(* CoDeSys 2.3 project: cy-wg-021-003.pro *)
(* Title: cy-wg-06 - ClevergyAS *)
(* Author: Andrea Ravasio *)
(* Libraries: Standard.lib 8.11.10 12:37:48, Util.lib 26.9.14 11:12:46, Visual.lib 8.11.10 12:37:48, WagoLibIdent.lib 25.2.13 13:49:34, WagoLibStatus.lib 8.11.10 12:37:48, SysLibFile.lib 8.11.10 12:37:48, SysLibRtc.lib 8.11.10 12:37:48, SysLibSockets.lib 5.5.11 09:22:24, SysLibEvent.lib 8.11.10 12:37:48, SysLibPlcCtrl.lib 8.11.10 12:37:48, SysLibCallback.lib 8.11.10 12:37:48, mod_com.lib 8.11.10 12:37:48, SerComm.lib 31.5.11 09:06:48, Serial_Interface_01.lib 22.4.13 12:50:14, Modb_l05.lib 13.5.15 10:30:08, Ethernet.lib 8.11.10 12:37:48, MBus_03.lib 9.2.13 17:51:58, WagoLibModbus_IP_01.lib 26.5.15 11:20:08, WagoLibMBX_01.lib 20.3.12 16:32:38, LON_01.lib 28.9.12 14:05:10 *)

(* PLC configuration (modules and I/O channels)
0750-9999/0545-0008 8 DO/DI Generic [Type_34_8_Channels] node 0, in %IB56 out %QB32 {INTTypePAAssignment = PLC; INTTypeModule = plugged}
  VPN_ST2 AT %IX28.0 [BOOLOnX_I] I 1: Digital Input
  LAMP_AL AT %QX16.0 [BOOLOnX_Q] I 2: Digital Input
  KEY_QE_ST AT %IX28.1 [BOOLOnX_I] I 3: Digital Input
  CIR03_EN AT %QX16.1 [BOOLOnX_Q] I 4: Digital Input
  CIR03_AL AT %IX28.2 [BOOLOnX_I] I 5: Digital Input
  CIRD06_B_EN AT %QX16.2 [BOOLOnX_Q] I 6: Digital Input
  CIR03_ST AT %IX28.3 [BOOLOnX_I] I 7: Digital Input
  CIRD06_A_EN AT %QX16.3 [BOOLOnX_Q] I 8: Digital Input
  CIR03_AUTO AT %IX28.4 [BOOLOnX_I] O 0: Digital Output
  AT %QX16.4 [BOOLOnX_Q] O 1: Digital Output
  CIRD06_B_AL AT %IX28.5 [BOOLOnX_I] O 2: Digital Output
  AT %QX16.5 [BOOLOnX_Q] O 3: Digital Output
  CIRD06_B_ST AT %IX28.6 [BOOLOnX_I] O 4: Digital Output
  AT %QX16.6 [BOOLOnX_Q] O 5: Digital Output
  CIRD06_B_AUTO AT %IX28.7 [BOOLOnX_I] O 6: Digital Output
  AT %QX16.7 [BOOLOnX_Q] O 7: Digital Output
0750-9999/0400-0008 8 DI Generic [Type_1_8_Channels] node 1, in %IB56 out %QB32 {INTTypePAAssignment = PLC; INTTypeModule = plugged}
  CIRD06_A_AL AT %IX28.8 [BOOLOnX_I] I 1: Digital Input
  CTL02_ST AT %IX28.9 [BOOLOnX_I] I 2: Digital Input
  CIRD06_A_ST AT %IX28.10 [BOOLOnX_I] I 3: Digital Input
  ALARM_PB02 AT %IX28.11 [BOOLOnX_I] I 4: Digital Input
  CIRD06_A_AUTO AT %IX28.12 [BOOLOnX_I] I 5: Digital Input
  CIR01_AL AT %IX28.13 [BOOLOnX_I] I 6: Digital Input
  CTL01_ST AT %IX28.14 [BOOLOnX_I] I 7: Digital Input
  CIR01_AUTO AT %IX28.15 [BOOLOnX_I] I 8: Digital Input
0750-9999/0400-0008 8 DI Generic [Type_1_8_Channels] node 2, in %IB57 out %QB33 {INTTypePAAssignment = PLC; INTTypeModule = plugged}
  CIR02_AL AT %IX29.0 [BOOLOnX_I] I 1: Digital Input
  CIRD01_B_AL AT %IX29.1 [BOOLOnX_I] I 2: Digital Input
  CIR02_AUTO AT %IX29.2 [BOOLOnX_I] I 3: Digital Input
  CIRD01_B_AUTO AT %IX29.3 [BOOLOnX_I] I 4: Digital Input
  CIRD01_A_AL AT %IX29.4 [BOOLOnX_I] I 5: Digital Input
  CIRD02_A_AL AT %IX29.5 [BOOLOnX_I] I 6: Digital Input
  CIRD01_A_AUTO AT %IX29.6 [BOOLOnX_I] I 7: Digital Input
  CIRD02_A_AUTO AT %IX29.7 [BOOLOnX_I] I 8: Digital Input
0750-9999/0400-0008 8 DI Generic [Type_1_8_Channels] node 3, in %IB58 out %QB33 {INTTypePAAssignment = PLC; INTTypeModule = plugged}
  CIRD02_B_AL AT %IX29.8 [BOOLOnX_I] Ch_1 Digital input
  CIRD03_B_AL AT %IX29.9 [BOOLOnX_I] Ch_2 Digital input
  CIRD02_B_AUTO AT %IX29.10 [BOOLOnX_I] Ch_3 Digital input
  CIRD03_B_AUTO AT %IX29.11 [BOOLOnX_I] Ch_4 Digital input
  CIRD03_A_AL AT %IX29.12 [BOOLOnX_I] Ch_5 Digital input
  CIRD04_A_AL AT %IX29.13 [BOOLOnX_I] Ch_6 Digital input
  CIRD03_A_AUTO AT %IX29.14 [BOOLOnX_I] Ch_7 Digital input
  CIRD04_A_AUTO AT %IX29.15 [BOOLOnX_I] Ch_8 Digital input
0750-9999/0400-0008 8 DI Generic [Type_1_8_Channels] node 4, in %IB59 out %QB33 {INTTypePAAssignment = PLC; INTTypeModule = plugged}
  CIRD04_B_AL AT %IX30.0 [BOOLOnX_I] I 1: Digital Input
  CIRD05_B_AL AT %IX30.1 [BOOLOnX_I] I 2: Digital Input
  CIRD04_B_AUTO AT %IX30.2 [BOOLOnX_I] I 3: Digital Input
  CIRD05_B_AUTO AT %IX30.3 [BOOLOnX_I] I 4: Digital Input
  CIRD05_A_AL AT %IX30.4 [BOOLOnX_I] I 5: Digital Input
  ALARM_PB01 AT %IX30.5 [BOOLOnX_I] I 6: Digital Input
  CIRD05_A_AUTO AT %IX30.6 [BOOLOnX_I] I 7: Digital Input
  AT %IX30.7 [BOOLOnX_I] I 8: Digital Input
0753-0648 LON-FTT [Type_55_1_Channels] node 5, in %IB52 out %QB32 {INTTypePAAssignment = PLC; INTTypeModule = plugged; DataStream = 1F8B0800000000000400ED5D7B6FDACAB6FFFF4AF73BCC41BA47AD141A0C84909C245B144C83368F1C1EE9AEDA0A393080778DCDF12369CEA7BF6B666C63E3F18B47D2504B5BDDC41EAF596B66CD6F3D66797CF5C7CFA5821EB16EC89A7A9D133E147208AB136D2AABF3EB9C65CEF24225F7C7CDFFFECF555B535BAA89F599; DataStream = 34C1081E528DCB9F867C9D5B98E6EAF2F4F4E9E9E9C353E983A6CF4F8B858270FA57A73D982CF052CACBAA614AEA04E7DCA7A6F14FE5D09DAECD7569D982C61785CB42E1F21CFE3DBB2C089785CA65A10C3F72E82F79D69596F83A272A78895553D2F1B82DC9AA3C160B173934C0CAACA14D2C7ACB0401EBDA92FCBECED5A6; DataStream = 53F4AC593A9AB02B68817560B08B2D5D539BB2BE7C0252F7EEA85CD0AE06D223BE93CCC575AE7EF9ED936C7E9B3CE70B4235FF3447EF1AD8C0EA7F2555437792820D5397D0BDAC2812EA482AD09751AD20D4DF7F6BF7BA39D4D1A69682BBD6F201EB403C07A38B1019DF8EA4FFE83DFC8D27A641AF6D5EB52FC2E5215EAE14; DataStream = C9C4AD29213E93B1EEDE83BB64E85AD39B4201F1FEBB3AB5EF7B9E184CB415BE815BEC87E7CE9FF8995C27FFF35C6DA953FCF346B83A653F5CBE4E231873992653763368DE0D556D8A9964EB07E94DF7116E537F939E2ECF655552B84D7D37DD475A465B9BFCC0D31B53B730C8E0FCE96900D336954C4D7F76DBACAF789AF5; DataStream = 5644AD24E5662629066DE65E715B7530996836DD64287D7FBBAD6C0DAE6B1668232CAC4B5556AE73A4F31C3AF50C08369F34FDC7BDA4CBD203289A775236EE796EC569CC765A13AD39AEF65C1437D5C7A342E4A65F8762F588A34BDDFBE1587BF87BACE3FF58B0F842B469AD51EAA3DC779A069BF894C6DB94AB4D89342A85; DataStream = 5625D7ACA0760921DA455B26D33046545607589D0EE5259D5AEF9FFE76D24F5F3BCF9F9BEDFA7882E547EC69EABDB221FC9D2E6BBA6C3EAF8577AFF85A0EB0FE284FF0F01934AF36F9A16A4F0A9ECEF114B4D173C7F74843D6011960206F5AEACA82495D5FF0B30C2670264FC8DCDC74351598F05EF135AD6BEA4C9E5B3A35; DataStream = 31B04A565837656C6C0E6ACB70BBDA5096CDEBBEC73E3E9B7820FF17DF94AE4EDDDF9E557F1ABEEC7F594428452142699F8800AE8769190900411BD82D63F1C06DF9CBC341318383E470D0B3CCB7850795A3C183F3283C38DF1B1ECC6405131721897BD084B67DD234DE3D709BEE110F5C458F07048764023C38CBF0E078DD; DataStream = 03A1783C78508EC283F25EF120B98340D63931FD495C8475DB5F1E142A19281CB193503C3F1A54B808A4A1D808B1A8A1B0575458694920819AFE3B2D49D0B06EFACB03C2790608C7EB25A40D1A0277D619C75896AF4E79D9EBED52DAD109EABC1092A1CEA74C51D345792FEBA625296866A913B65AD0830283BA99794E9546; DataStream = 8E58AB591E3919FEFF7A7964686E278785581B10249EC012B8EAB0475390268314A666B465660BD0AFE61CBAE26529653642AF975286D62C519C021A8CE499E50C19DE1032BCBE979812188E27B75C8DCA2555F7964B3241B5C8F25DAE92000351C4014EEA34786967C8705CC8F0F67C86E3492855AB51D050DD1734488AA4; DataStream = 2F93A0428D344C880936D10C0E8E0B0EDE9CA350BCC8E0E0907090DC4BC810E12811E1ED3908C70409515985EADEB20A24ECC789928DCA33C929E0849060D3CD20E1B820E1ED39094703084221CA49A077F703098B4769325E6AD344B0D0B8FD3C86494E9152F090CFD0E1B8D0E1ED390CC211C1C359243C9CED2DDD0857C6; DataStream = 89528D041B6A1393344C9A6EB46967C0705CC090B90D192EF87101FC853B4D5613EF4364C07094C0F0F63C860C190E8F0C99C7F0DB0343E631BC5E3D53142C5CEC0D158C27D99C2C92A042BDD920A820AA49738F36E50C138E0B1332672103051F287CCA40E1B70785CC51C87624D820F9BD05B22991ED48FCEEE8F0F65C86; DataStream = 6C47E280F905820D5972E1B74785CC67C84021E03064DB111930BC3D77214386C32343E631FCF6C090790CD9D90B6C90FC672F14B3B3177E7B6C787B4E4376F6C20B9CBD90021AB2B3178E1319DE9CD7909DBDF012672F244486ECEC85E34586B7E73364672F1CF465EB849890BD697D9470F0E61C85637AD1FA578483E45E; DataStream = 4286084789086FCF41382648F845CF5E480809D9D90B4709096FCF49381A40F8352B1D3D672F244486ACD2F168D1E1ED390C59A5E3CB9CBD9034DD98952E1C2530646E43860BFCB3173260F8AD81E1ED790C1932BCCCD90B1930FCD6C090790CD96BD681B31792E61EB3D7AC8F12133267210385E0D90B1928FCD6A090390A; DataStream = D98E041BA4E0D90BD98EC4EF8E0E6FCF65C876245EE0EC852CB9F05BA342E63364A0C03F7B210386DF1A18DE9EBB9021C3CB9CBD9001C36F0D0C47EF3104EE18EB5B713C5F9DB635B523E93F7A0F7F036BF4EAC635E3E6EA1F5FEB8DDAB0F6F5EA8F9F4B053D62DD006AD739E1432187B03A810153E7D739CB9CE5854AEE8F; DataStream = 9BABBA644A8A36BFB96ACA0A462D03FE67621D4FE1911C6AC0CD7B974499D020CDC8145EE7C8BFF0B7A62F25D36D54216D3AD2DF9AEE792E87EE2473719DAB5F7E23B0A54B4B4AC640EF7E562BEFBF81089F61488C6F84A2F16D30AC751BB57EE3C3F0CB1D3C4971EE3A17028439D4C733E0579DE0C856F47D4CF28225F053; DataStream = 3C154AA7C582504442F5B258B8148AB99B4DB8A6AC70AFA28F92618FC00056EAC4FC5AF99E43740983F83944D1F33A775ECA21024BD7393AB0F6911070EDD1640F131C0309C5F160D81FD5874C52181A184D79C29EA4583783C7C989123944B48CB09F43235586CEFEA998FF6AA98F92224F9161EA30B1D08DA159FA04FF73; DataStream = 6EFE8B2F94877D51B596C8214FB81B9B64EE7ECA4B6B4945019061BFF382234C3F5C0EB13BEAF0A470451FC873D5562C5B144792996788900A4F193944B8C36C31D8437A46403146A6916AD05E40A7E63017464B35F11CEBB4AF963198907768E81F6B39CFCE4A678E78B4279E70A3EEA0F5A92B36C6ED5EF7530EF5663303; DataStream = 9B945050609911219DE19A47DCA24F5CBBD5A125B2211D91578C358B3B7121B295F89349C98D5D72E1522E6545910D3CD1D4A991484E98E9AFA5F55A72175003B402AC3CD104244DA7A0E3065F8C56AFBB66FF8CC7FE9468B94B83317CE630ECE090DB49C2F55F5CF35C7478AE3112C8248F01F09AFA73D4DA8F649AB0633A; DataStream = DC961C6E793D24D5A5C1422314932853A9E4C1815229201F3502113A35B8EDF5E3046444029AE4C24335FF209BC8B299478078CC413AECCAF10FB09C12192A5B218350091375D371A06ED436F6C9362DD6838ACDBCAA4D71D49A4AA49F861ABE940C4E3F07D052C1A3A4C25BD2D18FB2E94ECE864036F8694B495679EC7F6C; DataStream = 0D9B31FA36B51F0E67DB9D28D634B55542E7888A00FF786CA22DD0B957A0E2B923521794614B8154FA68B83854CF541A69A511A21C10A2EC0A51F60AE131AB80B768429AC48B72CEB7A4D42644C842C540DA0C91A6324E6644B79668A84BAA21D190873A0B7ABC5C55EE42F939B61F0F178D3680D183C94A0BE62940A17876; DataStream = E687BB342070C1453A9B4CB864AC8557057700EEF3EFDEA5C458F8A46BD66A67C89EAFC2217BEEEB6167008B4361BF4A6D85BD0F9AA660493D046C55D62A047D6EC9BF411F4D00C26CE859F3DFDE74303E46AA6540DB998C95E996A25894449428719174664A3253E203E09D2DC99C51D94D25F9A6651B83B39DCB6D03BC65; DataStream = 2EC8A6C08445E81A1771C206472870235E2039D622D1273DE66F239B93E34E2B15372FB4026229A4DAC171287FF7AE50272359F66524D94994DB26249DA7EDF8F57CFF3949D6832F252908DC9CE4205492B094E49AFBC88C246B169E90AC1C3E09D175919B701492F74A9E9A648660ACCDC636B9F054846D900E2DE0002B78; DataStream = 62520BAF4447E909B293864D6CCC88ED2D034B32931159BE6DB391D2547739DB5B56DF86809044EA449757A6C635C8890287A987C4BE39AFE9BAF4FC55A87C27EADE643334D390442E23CCB64AD71E2FD96A31E8231EBC769FE20958EBF76B5F62E4A3D0C308D8885071C4637C006B42054D16920E0E0ED6132489E9EAA8C3; DataStream = 03096D0F01530FCA15AB01E136878433976CC9D46F6BFDB5C045AEAD7525FE2A9C7DDF583361E8C8925DB541BDD55A0FC5F6468BF6F36F4B9A2674C684F279B95AAA94CFE362337B18FE3DAA353CC3C045464E8CB6217DD935D2CF662A0F7A4B641CC6A52DFD80584C133A275EB37B7544624133F1768867FBE662BFF0C3D0; DataStream = 8785CEA8D508411F2EF8B80F6D0B3E2C901ECB5347B620F65410D3BEC3C638A1E2EFEAD8BB127E0D604DB26CFA0B0537958D9150B03A3717BB8700B6FC0EB9F00110BB48285F14AA79C149AF38CFFC7299525290B09F54E9FEE3B8F84D8750A9B80E66DAFD873411FA0E302B78B6F884750D4AB5E40D91307A04E738DAF70B; DataStream = 09F9E831839CCD4AE242CB8FF2D4921444162C5DA77BC819337609C54278EA28C82B3C50D84FCE203C3119C3AF90925FE130FC1693F25B4CC96FF130FC9692F25B4AC96FE930FC9693F25B4EC96FF930FC9E25E5F72C25BF6787E1B79294DF4A4A7E2B87E1F73C29BFE729F93DDF23BFC938ACC627EBB9AE0D3C5B7D65F0BD; DataStream = D89EF58B57C66121C2D0C5F12E1CC8E825066521C2EAC5327F200B9818A185081318CBFC81CC6162B81622EC612CF307B28D89B15B88308EB1CC1FC85026067221C252C6329FD86AEEADEACF8908DC2C0C298847F493435BC403EBEF1539DCBB1B40CF58D24FD05253CDC5099A4ACF2768A159E48AAC5A263E41AC203861D6; DataStream = 3479E6AC542055FE9CCDA12F58E2473CDE1C5A50CC67FA58543AB0E895384D3A3055FCEA88D121039A267EE506E54B46255CF768830309535A27CA246E31749828DC487C2A45563CC0ED0389517483EA5B50EC34729479722C28917041C8FD03497276E16A175D9C3BD7C82E6D3211FA455B1C5C9E01039914F2700B876CAC; DataStream = 8ACA61795E6FD8257FE3C9930BEB1DFBAABBF543BF14B3FD963DFD728C0B5C07C998B735BBFE2345C2DC7926225F1E1448711F7ADD1C7998C03BAE2147BC74097222F0CEF9F12DF7A9D8AB8721DB1E69DE8ED02821B6FD11BA61C51A25DEBBA7F52454FDC7642BCC574E522AFA3C86927FB19921DB6FACA624B26E6DDD5FD4; DataStream = 26AAE476135E61729E54C4955DA83456F023569254CDB8A54DF4897849B9656CFE6EA3A45DF9BA0B97B8FA422FF911A0E8DEA7A9A7E16E68513D1C9BDA98E06C94DECAEB4ED144B20C02B6362CC7CACB70B64C71F69EA4D84340B6CC03D97BB67716BB23C9DFC6B177DE3676C05DA82DBF08D472654EB195C3055A2A192D93; DataStream = 8908C55E16565910131DB784692717513951CC1B085D042EA8BECDD845E0C2E61B0C5EF8C5436F347AE19700BDE1F0A5C8DF834F15BFEC1BCD2E2E3C33E4BE0A9EA6A2891BF82FBDB4F6F6F6B9D7C432FF4F9197E061A730B49EC712985B7EB916F31C6D1AAF6B74234621855E46F8C794F46E06788790DB5FCE6B3B9F17AE; DataStream = F9A5B5962BCD90C3E2D32445F2F07C204A5D91F3CFB07EE2D4F31CBE38B28FA5E9E967F0BD8940B4F3D85249CE2B464FE395199311753595565793A95BBFA778F8632E5C2113D46AF971869B97038143ABB45C9059BF57B5AE09DDBB4EBA8E941D686F7F940CC4CE63CF692CBEE3245A8D1397F22F943078C12C814D987716; DataStream = 4EB1CC0DA1E327C41F42738DB4BFDBA8105AF375171E429348754745F46C1E15D7BB4717A50DC9B74E48124DF4BF4254F12AA2FDE2CD4C91E6C9CDDCD168636CB1869DB3CDB71A7488E23722B98A27332A7CDEF7B0952A2413C251E73D48B25E432F5FCAD1900D4264BA8B1C539BC6AB9473F42C33AFCDF2D42B33769142B3; DataStream = 4CF2821923F42AC51DBD1556F313599F58F24E7AA5019DB14DE7550A3DEC3931D8C9897B98149BD2AB147E74F06421A932749C9F4996B2D3CC2C5D5A634AEB558A419A184F1FA4C90F1047562C7DA7F999D9B4C636AD172AFBEB3D623DAF4BEA3C29F3DC905C032A634AE5552CC908ECEA1EA4B00899438A11634144F2EEAA; DataStream = 9E7A7D7065C12EAD43AE8F188B3252098DBCA9E5975832922F9090D921C4C84E8B4DEC552C4B5D5B2E2DD53EEAC048B9F0B9724D80E201167D721BD384BEF1146C8C32CB9BC91D31AE30448E31A134360FE687C595173A72E46535BF221C92C3877690C915672CAB6387E0ABD81B7612711E4CF92EF22894CA987F78E7216C; DataStream = 4C47522DC0B489A69ABAA624649D9B9359524A639BD22B452D2BF0C9D8D6FD0E92802A3935392F6F68980CC468EBF23429788589E19079150BD3C72B4D37F34BC9F8B18B183A253326645EC5AA381CC9EA3C4F3E90B58B2CAB352DFAB1AD57B1295E81884DD8974084D6AB5815BA19925735539E3DE7A7E9427DAE546C0B84; DataStream = 111C1F36EE8FB12A7D6CF0DFF74DB470E01EE0F172A5E0E89DD32D8EE8AB22AF69714B21499FFA239E26786D83BBC5E679FE10A76FED90E85FBF834D3FA2B9455AD5B01FDCC83FD252179655C507D9355C97AD84561B6DEE1086971AD993E2BC23F19165DC3726E8FFE8914896A238E56BB17A35D8E54C61FF615351678D6C; DataStream = D67F841D3F1573D8882B286D4BCFB7DBF17C153B3DEE6C119C252C7C299E577CE7D114CF4B82BBB5483ED942F61E68EC92FA1D0BCFA75CFC83E14C7B31EAB58B29064F1C1BA88E1543B6926C31D25D1EFA154AD33310559F2273E7FCF6BE5647CB900304C2CE18F37FF3326A8A5DF2115B3AE5D0D9376EAE3CEDFD7FA1F597; DataStream = 1386D2DC3EEB67BDC17573C52AEB7C0979642FE1A044CDFEB83B6AE7505F7AA26DD8109DFAA90C0875D594250549930989BD744CF6AEB9E47A7762773CEC8D0762B79180D213D9DF8D21D517EB62EB5EF4721964B2AE680646920AE02E3D62FBE8312ED97ABB3710C7CD56DB47B11841718A892D8CA7D910DBE23048BA1420; DataStream = DDA74776029B53FA491A4D7F76BE27C0A5DE68C1100C7BFD2FB0EE7A7F8EEEBCC4CB41E2C0B2B64C3955E37ECD4BF52C866A8A69DBA0CC0ED83BF5683457BD2B5EF576CF0D4CABDD8304DA4DCB424C72BCE90CEBC8B0A88060864208FED51441C43F03641AEE4C2A9AF6831CF91B4789CD25A515A5D8A2AE6B3A22A770AEB0; DataStream = 4ABC9650351CB0A16FD65AED68CD76494E37988EE654ECF7A3D5DA3F94B28AD6B995F0B11C751B62FF33A9A38A526A9765A2CF300AA744036346A3D5DB6439A8D67E96C94B905344F3285C8AC35647EC8D869B642B01B29F65582D4FC8A07837C10813F643887E6E751BBDCF9B34CF0334370E6575138C5CA2B5D1F0769364; DataStream = 354892AD6666A83413747645C266CC470CA05AAF8B83014C59ED7E43C92E6200E3013F6B80A4628F7B2A02901E88E29FE356F7BED626DBF69E055108CE99DDFA73ADC5F53AFDF73DA48464D8736E638FEF1D133F0BA3D594F870EEFC2E402B3177826BEDF1AD580315F7C35070F16C929C699A194AB2D9EB0D374906D77903; DataStream = 3F58737ABC20F9A01791F01D99654965AF29BC0F21DE103F8E3EF9690761A9E5A16A31D613116F759B3D3FEDE0040F9E0DF021D3333EF832188A9D6017C1F5395CD8674B23D94076AD410851D0C891C8D3CC7C104D7C642570F155305DAA7D88523219EABD2EF95A9A4F71F3413C243D4D31DD4286AEB4D94C91552E1600C9; DataStream = 5EB3D96E757D2E493EA87FAC389414D7CA6C5255F2A53F18F9A5F40CCB174DA1A5A951A93C1B260E0C2140E785A44F9F24B277C2AE858938EAFED9ED7DEEFAF8092AAF63DD3DEF54D9C3286D704A916B8527E41B96D3B04EE31D81AE863629AF486641E55A0342B24766ABD11AD263613797B3EAB294926CADDDF1D28DF20D; DataStream = 869A2929A74E2D012D047D24BE35ED4F40EF481A4753A12B5A6106C6DE404E63982F72069D895509D0266CD486BDE178705FA73C09D14E45242FDC0DF20DFAC568E722923E775B64837E29DAC3B08BA3C16ADB05D26CD2142CE9881BF203F936D8ED766708EE7FDF3F3C416888221F363A5EF2C5688783915FC8F3450AF66F; DataStream = 5B9F6EF9FC73BC8FA80EC204F075508CF145B8031437F201C50C3A227CC271631ED0488E9D0A1993D8E10E30CDB1AF21B463473AC87770A9360109364129CCD168F509491F419EE30F0401D5F2C989DEF5C500E1E0A22484F33A261F1B9E829BAE590FE0AEBFA3F50FEF137533EC7FF4E1BEC00B013C7D80074C10C6D0E8F7; DataStream = 3B1CC07E873FCC3F9C8091D165F587028102417023C2C491AE07A3BB7B5FD7C155EB178FEC7053573CF9280EC5C130308CC1C51BD24FBA19A37DF1A62DB8967DFD2D592A0E61F551D63595BC6F02B84D4C13560DE644B0178821B49B2CF8B187CD82D8BDAFF73A77E34EED2F1F07C145EFE3407A508923A980D55859662261; DataStream = 3BBD6E6BD8EB5343ECB37B9C70C42FAC6B53611AB11E66E4691FB55697CC9ED8F7797B454E8E827CD11749AB95E2B85DA10125A15D1BC2BF10FCF5FCF17A90F51E44943AA3153B2A417A413E193DF00169A2228EE2E75ABFDBEAFA228D5231598856B543B4C03BF22933447749F29F6DED8914D1B095B2DA78C79E4BB32DDE; DataStream = 8BED7170BCDD5B5C13E1BD1BE5F5B9EDB8C6C07B37CA5FBB05D3B29558A5683FAD2DCF301A48330CC4A85DA096CC40EF3ED6EAE47060F7908222173CEF363C91A04DB863DFD17E4ED44929AC9362B4BB46890E3CC680D9E300FD7218FD52B4BF46E90F99413B6DD2DAC0770DD95829D2F3FB602F6761BD94A39D36DACB1DC0; DataStream = 13E5FE04D16D893AC99C4D004F44080956048EC384AB84755B8976E568376133520D235A8D76E3C278EF0FBB274C07E057D4200A8550852BC4387AB46F4A5E6158E02C175E37A1A32654383E5F2CD4117628D6055E664A8975FD7F27C03A91D664DA2F4ED1CD0F1D2FB547B8E21605F129F7FA9D5A9B9315373CF4429E6DB4; DataStream = 06B58F6DB1118D7AAC30C8E1CC79D3884B7074D7A80DC9CE7A6D381A44A3E01DD64992C925EB941A86501E88ED267584A231D0CEE549BE239EA258ADB56BFD4E34ECD9F2DBEF5191A382587113976C5FBCEBF587E0610CFE8CC6B99E5332163943BD7BB0FEAD86188D693EDD09A12476C95447A356DFD6383625318AD7EFDC; DataStream = 73D90BA2529D86AA49F4A7DE166B7D8EFA0441C947D32EFF8B201998660ED6D8A3C874875613C9CEE9585CCA9426ACBF61ABF9C51EDE06076778AB72BB3EB8CB95B3C9E4439219CD37915A4FE4D67A72BBEAD4BA2392061DF6FD715B7091053B2050452B2BA23AE88B9D1EACB840079C3D27D681A75A8D54A8D0B41E136326; DataStream = CF2D1BAC57CC29A1DF61E4767BD7EF7DEAD7FC931F5C8E4C9F680D56DEA9C1A23569E89DBF308B6B635C3DEB8B03D1BFF5C159AD3FF1C402EAAC3377DB01248C5CC041D2C105CCA400089490A2CD23396DF77CFE3F27966C6B12C4AC0B771ED6A95EB2C338A8DF0DC90DF6CDB190AEDABD5A833B019C5D2B4BA59D4D2C5D07; DataStream = EF42213BA3D214FAB27BFF805A331F374F92811692C2623FA2DFCAF30934900DF4242B24A635C0A223DD52D9DEADAE2DD9E3E4B57D92BA5F3FFF216CC4475D1EF39C48F416E8C4703F74395BD95573FEB1A5A549C4EC4BE43BEF4C2BC0C7825121697F72C32B96F7512ADA13C47F18816D8A17EBB6D61E72E5E2997EE04B8F; DataStream = 166D3DB40F782ED3D10E1D50B0DFB53EBFF3208E8D54C5D1C0B0BEC36C7B374CF18A1C3463CBD1A01DA9F8A749960E7575B595E311BE239B3C76D11FF17D4F600518B4FC10EE9EB007D003791BE0046173F2E13D59CD71FAB039F94B0BFCDB078CFEF91F4B33FF254F15CC7E911D03F68BCDAB7D956C094D26786532A5B7B5; DataStream = E404692415F0241B4C1B88CE004D79AE6A3AA884AF5B1D9B96AE1A841287BEAD913393242AE818D12F92CE7CDD85796B43F18E3BFCE584AE77D976BDED0A33BEC3FD18E67093A82181CB5D67E68AA41525CBD428010223E4336CEA1C93BD73F30963D597FF21F93BAEA9A19DD646C35E101DB0442B263455E1161AD1276FC5; DataStream = DA30DA0FAFADB9C8DB503C017658CAE789D454F3EB4828F94EBFFB69FCB9DFF1D730716AAF344D89E5B5DEEBB5A3FD702EAFAA3C5F400467E9F388596B7DBA058018F53F89D15E39B70792579D687C0F84922759D44DEE39CEC05A31C816A7EDD6B071B1CC9565862B40AFD98CF1D5DDF8F901138224E6E1A75E29BDCD9027; DataStream = 68F345583C73F0209E492D84C94A4ADED19F2B6BB9E2BA2B94B2D811FB9F026AC7D91E92DD516049450C203393C05A037890A21DAEEF4ABB68D6BAE35EB7FD25C695B755EE493617343B4D52FC1AEBD436DFE13DF4C5E084727CFBD604E797D20FD20DAB200DA1D7AA8B312EBC5DDF4A073B965CA7F6577061733C76185B6D; DataStream = 09FA4B90E2948C473459B1DEEBF63A5F62DCF4065E584B79EA8618D1341BE2EDA8B35101145C757500DE073D01B97AADDDFAD887083BC6EF5E6BEF245E6CAAB181D9E6AC319728AC2D307409A882C5AAC56DE6B853CA588898F3008FFC54DDF8F6BE4E7DE470ABE03688749E1974F6A269B9F703AEACDF1E9FFA4BA04F49A5; DataStream = DECD15ADD76B19F03F7008ECDAEB06041AF75837A021D1960F408D346345DDCD1544054D5A47E4B639234D3AD2DF9AEE790C1896CC05E8D6E5379B734AC540EF7E562BEFBFB535F5B3A6FF30BED102ED6FA446A751EB373E34EFEC1AB41630532820DE7F202B9E01BB105F45B6221F7018904F3090E5792A944E8B05A18884; DataStream = EA65B17009EB15A4B754EAEB490AF4483FF7CCB9E67A2F4EAD3BF94E1EEAB9419DAC4EE495A4849C5A300081C827EFECF681027C18FC0E785C12A91A65EF1560726016FBA8B5A7D3CD8394823DA98F72DFB94B06D5733856B0EE3FA6DBCD03B5C2D33BEAA3E67C5CDCDB6989DBA9BF13F7651EAA84D1929126209DAF93F324; DataStream = 9D547C9D44CA415A1059FC9D94137472EEEB647D265EA82877DAC678D92B36A07CBC6BEBD57B5A271B99DAFCE6FB77F8A34DDE8580653C9326F8E6FF010020230C50320100; DataStream = .; DataStream = .; DataStream = .; DataStream = .; DataStream = .; DataStream = .; DataStream = .; DataStream = .; DataStream = .; DataStream = .; DataStream = .; DataStream = .; DataStream = .; DataStream = .; DataStream = .; DataStream = .; DataStream = .; DataStream = .; DataStream = .; DataStream = .; DataStream = .; DataStream = .; DataStream = .; DataStream = .; DataStream = .; DataStream = .; DataStream = .; DataStream = .; DataStream = .; DataStream = .; DataStream = .; DataStream = .; DataStream = .; DataStream = .; DataStream = .; DataStream = .; DataStream = .; DataStream = .; DataStream = .; DataStream = .; DataStream = .; DataStream = .; DataStream = .; DataStream = .; DataStream = .; DataStream = .; DataStream = .; DataStream = .; DataStream = .; DataStream = .; DataStream = .; DataStream = .; DataStream = .; DataStream = .; DataStream = .; DataStream = .; DataStream = .; DataStream = .; DataStream = .; DataStream = .; DataStream = .; DataStream = .; DataStream = .; DataStream = .; DataStream = .; DataStream = .; DataStream = .; DataStream = .; DataStream = .; DataStream = .; DataStream = .; DataStream = .; DataStream = .; DataStream = .; DataStream = .; DataStream = .; DataStream = .; DataStream = .; DataStream = .; DataStream = .; DataStream = .; DataStream = .; DataStream = .; DataStream = .; DataStream = .; DataStream = .; DataStream = .; DataStream = .; DataStream = .; DataStream = .; DataStream = .; DataStream = .; DataStream = .; DataStream = .; DataStream = .; DataStream = .; DataStream = .; DataStream = .; DataStream = .; DataStream = .; DataStream = .; DataStream = .; DataStream = .; DataStream = .; DataStream = .; DataStream = .; DataStream = .; DataStream = .; DataStream = .; DataStream = .; DataStream = .; DataStream = .; DataStream = .; DataStream = .; DataStream = .; DataStream = .; DataStream = .; DataStream = .; DataStream = .; DataStream = .; DataStream = .; DataStream = .; DataStream = .; DataStream = .; DataStream = .; DataStream = .; DataStream = .; DataStream = .; DataStream = .; DataStream = .; DataStream = .; DataStream = .; DataStream = .; DataStream = .; DataStream = .; DataStream = .; DataStream = .; DataStream = .}
  AT %IB0 [BYTEOnB_I] First Byte of 24
  AT %QB0 [BYTEOnB_Q] First Byte of 24
0750-0464#04 2/4 AI RTD / ADJ./ HA [Type_44_4_Channels] node 6, in %IB52 out %QB32 {INTTypePAAssignment = PLC; INTTypeModule = plugged}
  S01 AT %IW12 [INTOnW_I] Channel 1
  S02 AT %IW13 [INTOnW_I] Channel 2
  S03 AT %IW14 [INTOnW_I] Channel 3
  S04 AT %IW15 [INTOnW_I] Channel 4
0750-0464#04 2/4 AI RTD / ADJ./ HA [Type_44_4_Channels] node 7, in %IB76 out %QB56 {INTTypePAAssignment = PLC; INTTypeModule = plugged}
  S05 AT %IW16 [INTOnW_I] Channel 1
  AT %IW17 [INTOnW_I] Channel 2
  S06 AT %IW18 [INTOnW_I] Channel 3
  AT %IW19 [INTOnW_I] Channel 4
0750-0650/0003-0000#03 RS 232 C Interface (Adjustable), 3 Byte [Type_21_1_Channels] node 8, in %IB84 out %QB56 {INTTypePAAssignment = PLC; INTTypeModule = plugged}
  AT %IX20.0 [BOOLOnX_I] Transmission acknowledgement
  AT %IX20.1 [BOOLOnX_I] Reception request
  AT %IX20.2 [BOOLOnX_I] Initialization acknowledgement
  AT %IX20.3 [BOOLOnX_I] Input buffer is full
  AT %IX20.4 [BOOLOnX_I] Number of received characters Bit 0
  AT %IX20.5 [BOOLOnX_I] Number of received characters Bit 1
  AT %IX20.6 [BOOLOnX_I] Number of received characters Bit 2
  AT %IB41 [BYTEOnB_I] Input data Byte 0
  AT %IB42 [BYTEOnB_I] Input data Byte 1
  AT %IB43 [BYTEOnB_I] Input data Byte 2
  AT %QX12.0 [BOOLOnX_Q] Transmission request
  AT %QX12.1 [BOOLOnX_Q] Reception acknowledgement
  AT %QX12.2 [BOOLOnX_Q] Initialization request
  AT %QX12.4 [BOOLOnX_Q] Number of characters Bit 0
  AT %QX12.5 [BOOLOnX_Q] Number of characters Bit 1
  AT %QX12.6 [BOOLOnX_Q] Number of characters Bit 2
  AT %QB25 [BYTEOnB_Q] Output data Byte 0
  AT %QB26 [BYTEOnB_Q] Output data Byte 1
  AT %QB27 [BYTEOnB_Q] Output data Byte 2
0750-0653/0003-0000#03 RS485 Interface (Adjustable), 3 Bytes [Type_21_1_Channels] node 9, in %IB92 out %QB56 {INTTypePAAssignment = PLC; INTTypeModule = plugged}
  AT %IX22.0 [BOOLOnX_I] Transmission acknowledgement
  AT %IX22.1 [BOOLOnX_I] Reception request
  AT %IX22.2 [BOOLOnX_I] Initialization acknowledgement
  AT %IX22.3 [BOOLOnX_I] Input buffer is full
  AT %IX22.4 [BOOLOnX_I] Number of received characters Bit 0
  AT %IX22.5 [BOOLOnX_I] Number of received characters Bit 1
  AT %IX22.6 [BOOLOnX_I] Number of received characters Bit 2
  AT %IB45 [BYTEOnB_I] Input data Byte 0
  AT %IB46 [BYTEOnB_I] Input data Byte 1
  AT %IB47 [BYTEOnB_I] Input data Byte 2
  AT %QX14.0 [BOOLOnX_Q] Transmission request
  AT %QX14.1 [BOOLOnX_Q] Reception acknowledgement
  AT %QX14.2 [BOOLOnX_Q] Initialization request
  AT %QX14.4 [BOOLOnX_Q] Number of characters Bit 0
  AT %QX14.5 [BOOLOnX_Q] Number of characters Bit 1
  AT %QX14.6 [BOOLOnX_Q] Number of characters Bit 2
  AT %QB29 [BYTEOnB_Q] Output data Byte 0
  AT %QB30 [BYTEOnB_Q] Output data Byte 1
  AT %QB31 [BYTEOnB_Q] Output data Byte 2
0750-0461/0000-0007 2 AI PT100 Resistor Measur. 10R-5k0 [Type_8_2_Channels] node 10, in %IB96 out %QB60 {INTTypePAAssignment = PLC; INTTypeModule = plugged}
  VRD03_ST AT %IW24 [WORDOnW_I] I 1: Analog Input
  VRD02_ST AT %IW25 [WORDOnW_I] I 2: Analog Input
0750-0461/0000-0007 2 AI PT100 Resistor Measur. 10R-5k0 [Type_8_2_Channels] node 11, in %IB100 out %QB64 {INTTypePAAssignment = PLC; INTTypeModule = plugged}
  VRD01_ST AT %IW26 [WORDOnW_I] I 1: Analog Input
  AT %IW27 [WORDOnW_I] I 2: Analog Input
0750-9999/0500-0002 2 DO Generic [Type_10_2_Channels] node 12, in %IB60 out %QB33 {INTTypePAAssignment = PLC; INTTypeModule = plugged}
  VRD03_OP AT %QX16.8 [BOOLOnX_Q] O 1: Digital Output
  VRD03_CL AT %QX16.9 [BOOLOnX_Q] O 2: Digital Output
0750-9999/0500-0002 2 DO Generic [Type_10_2_Channels] node 13, in %IB61 out %QB33 {INTTypePAAssignment = PLC; INTTypeModule = plugged}
  VRD02_OP AT %QX16.10 [BOOLOnX_Q] O 1: Digital Output
  VRD02_CL AT %QX16.11 [BOOLOnX_Q] O 2: Digital Output
0750-9999/0500-0002 2 DO Generic [Type_10_2_Channels] node 14, in %IB61 out %QX16.10 {INTTypePAAssignment = PLC; INTTypeModule = plugged}
  VRD01_OP AT %QX16.12 [BOOLOnX_Q] O 1: Digital Output
  VRD01_CL AT %QX16.13 [BOOLOnX_Q] O 2: Digital Output
Fieldbus variables [FB_VARS] node 1, in %IB0 out %QB0
Flag variables [FLAG_VARS] node 2, in %IB0 out %QB0
Modbus-Master [MB_MASTER] node 3, in %IB0 out %QB0
*)

(* Global variable list: Global_Constants *)
VAR_GLOBAL CONSTANT

	Plant_NAME			: STRING :='cySN:21 cyVER:1 - ';
	Plant_SN			: DWORD  :=21;	(* S/N Impianto di telecontrollo *)
	Plant_SW_VER		: WORD   :=2;		(* Versione SW installata *)


	(* Colour defines *)
	COLOR_RED			: DWORD	:= 16#2020F0;
	COLOR_YELLOW		: DWORD	:= 16#20F0F0;
	COLOR_GREEN			: DWORD	:= 16#20F020;
	COLOR_LIGHT_GREEN	: DWORD := 16#006000;

	(* Parameters *)
	Plant_DefaultTAmb	: INT	:=100;		(* [.1°C] Temperatura ambiente di default in caso di rottura sonda *)
	Plant_MaxRunTAmb	: INT   :=210; 		(* [.1°C] Temperatura ambiente massima funzionamento impianto *)
	Plant_AntiFreezeTAmb: INT   :=-40;		(* [.1°C] Antifreeze temperature, start circulators *)
	Plant_VRD_TAlarm	: INT   :=850; 		(* [.1°C] Temperatura di allarme VRD, blocco *)
	Plant_VRD_TMax		: INT   :=800; 		(* [.1°C] Setpoint massimo per uscita VRD *)
	Plant_VRD_TDefault	: INT	:=300;		(* [.1°C] Temperatura di default in caso di errore climatica *)
	Plant_CirOffDelay	: TIME	:=T#30m;	(* (Def.T#15m) Ritardo spegnimento pompe per ricircolo caldaia *)
	Plant_CirOnDelay	: TIME	:=T#15m;
	Plant_MaxWaterLoss	: WORD  :=2;		(* [lt/h] Massima perdita del circuito *)

	(* Filesystem *)
	FilesPath  			: STRING :='S:\';

	(* TCP Logger *)
	Logger_SERVER		: STRING:='';
	Logger_IP			: STRING:='192.168.100.3';
	Logger_PORT			: WORD  :=80;
	Logger_GETSTART		: STRING:='GET /cygmsrv/hsgm.ashx?';
	Logger_GETEND		: STRING:='$R$N$R$N';
	Logger_CHECK		: STRING:='True';
	Logger_CRLF			: STRING:='$R$N';
	Logger_DataFile		: STRING:='S:\LOG.DAT';
	Logger_DataFileOld	: STRING:='S:\LOG.BCK';
	Logger_IndexFile	: STRING:='S:\LOG.IDX';
	Logger_ConnRetries	: BYTE:=5;
	Logger_RecoverMsgs	: BYTE:=25;

	(* TCP Remote *)
	Remote_PORT			: WORD  :=10;
	Remote_WELCOME		: STRING:='Connected$R$N';
	Remote_OK			: STRING:='OK$R$N';
	Remote_ERROR		: STRING:='ERROR$R$N';

	(* TCP Sockets *)
	MAX_SEND_TCP_SERVER					 : DWORD:=3000;(*60000*)
	MAX_RECEIVE_TCP_SERVER				 : DWORD:=3000;
	MAX_RECEIVE_TCP_SERVER_SOCKET	 	 : DWORD:=1500;
	MAX_SEND_TCP_CLIENT					 : DWORD:=3000;(*15000*)
	MAX_RECEIVE_TCP_CLIENT				 : DWORD:=1500;
	MAX_RECEIVE_TCP_CLIENT_SOCKET		 : DWORD:=1500;
	MAX_RECEIVE_UDP_SERVER				 : INT  :=1472;
	MAX_RECEIVE_UDP_CLIENT				 : INT  :=1472;
	CONNECT_WATCHDOG_TIME				 : TIME :=t#10s;

END_VAR

VAR_GLOBAL
	TestNodoInterogato: BYTE;
	NodoDaInterrogare: BYTE;
	InibiscoModbus: BOOL;
END_VAR

(* Global variable list: Global_Retain *)
VAR_GLOBAL RETAIN PERSISTENT
	Mode_Manual : BOOL := FALSE;

	CAL01_Clima : typ_Clima;
	CAL02_Clima : typ_Clima;

	VRD01_Clima : typ_Clima;
	VRD02_Clima : typ_Clima;
	VRD03_Clima	: typ_Clima;

	Ctl01_Counter	:	DWORD;	(* Water counter *)
	Ctl02_Counter	:	DWORD;


	DelayAllarmeTemperaturaNonRaggiunta: INT;
	DeltaInterventoAllarmeTempeaturaNonRaggiuta: INT;
	OffsetSetPointManuale:INT;							(* Offset al Setpoint manuale per comensare lo scambiatore *)

	SogliaMinStartAntigelo: INT;
	SogliaMinStopAntigelo: INT;
	BitAbilitaAntigelo: BOOL:=TRUE;

	PercVelMin: INT:=75;
	PercVelMax: INT:=100;
	ErroreTempMax: INT:=100;
	ErroreTempMin: INT:=50;


END_VAR

(* Global variable list: Global_Variables *)
VAR_GLOBAL

	SYS    : typ_SYS;
	Logger : typ_Logger;

	Lamp	:	LAMP_AL_GENERALE;

	T_AMB	:	INT;		(* Environment temperature *)

	(**** PLANT OBJECTS ****)
	(*...*)
	(* Boiler *)
	CAL01	:	obj_CAL_VT100GC1B := (ID:=1);
	CAL02	:	obj_CAL_VT100GC1B := (ID:=2);

	(* Cascade *)
	CAS01	:	obj_CASCADE	:= (Tmonitor_On:=T#15m, Tmonitor_Off:=T#30m, DeltaTempThr:=100);

	(* Water counter - 2 PULSES/LITER *)
	CTL01	:	obj_CTL	:= (ID:=1, Peso:=1);
	CTL02	:	obj_CTL	:= (ID:=2, Peso:=1);

	(* Heat counter *)
	CTB01	:	obj_MBUS_CTB_SHARKY775 := (ID:=1, Address:=16#53104561);

	(* Cronothermostat *)
	THER01	:	obj_CRONTER := (ID:=1, Local_MaxRunTAmb:=250,Histeresys:=10);
	THER02	:	obj_CRONTER := (ID:=2, Local_MaxRunTAmb:=250,Histeresys:=10);
	THER03	:	obj_CRONTER := (ID:=3, Local_MaxRunTAmb:=250,Histeresys:=10);
	THER04	:	obj_CRONTER := (ID:=4, Local_MaxRunTAmb:=250,Histeresys:=10);
	THER05	:	obj_CRONTER := (ID:=5, Local_MaxRunTAmb:=250,Histeresys:=10);
	THER06	:	obj_CRONTER := (ID:=6, Local_MaxRunTAmb:=250,Histeresys:=10);
	THER07	:	obj_CRONTER := (ID:=7, Local_MaxRunTAmb:=250,Histeresys:=10);
	THER250	:	obj_CRONTER := (ID:=250, Local_MaxRunTAmb:=250,Histeresys:=10);

	CronEd	: 	obj_CRON_EDITOR;

	(* Valves *)
	VRD01	:	obj_VRD_POT_new := (ID:=1, fFeedback:=FALSE);
	VRD02	:	obj_VRD_POT_new := (ID:=2, fFeedback:=FALSE);
	VRD03	:	obj_VRD_POT_new := (ID:=3, fFeedback:=FALSE);

	(* ModBus Pumps *)
	CIR01	:	obj_MODBUS_CIR_DAB := (ID:=1, Address:=1, OnDelay:=T#1m, OffDelay:=T#30m);
	CIR02	:	obj_MODBUS_CIR_DAB := (ID:=2, Address:=2, OnDelay:=T#1m, OffDelay:=T#30m);

	(* ModBus Double pumps *)
	CIRD01	:	obj_MODBUS_CIR_DOPPIO_DAB := (ID:=1, Address1:=3, Address2:=4, OnDelay:=T#1m, OffDelay:=T#10m, Mode:=2);
	CIRD02	:	obj_MODBUS_CIR_DOPPIO_DAB := (ID:=2, Address1:=5, Address2:=6, OnDelay:=T#1m, OffDelay:=T#10m, Mode:=1);
	CIRD03	:	obj_MODBUS_CIR_DOPPIO_DAB := (ID:=3, Address1:=7, Address2:=8, OnDelay:=T#1m, OffDelay:=T#10m, Mode:=1);
	CIRD04	:	obj_MODBUS_CIR_DOPPIO_DAB := (ID:=4, Address1:=9, Address2:=10, OnDelay:=T#1m, OffDelay:=T#10m, Mode:=1);
	CIRD05	:	obj_MODBUS_CIR_DOPPIO_DAB := (ID:=5, Address1:=11, Address2:=12, OnDelay:=T#1m, OffDelay:=T#10m, Mode:=1);

	(* Pump *)
	CIR03	:	obj_CIR	:= (ID:=1, OnDelay:=T#1m);

	(* Double pumps *)
	CIRD06	:	obj_CIR_DOPPIO_new := (ID:=1, OnDelay:=T#1m, ExtStatus:=TRUE, Mode:=1);

	(* Temperature probes *)
	TPV01	:	obj_TPV := (ID:=1);
	TPV02	:	obj_TPV := (ID:=2, IN_WMIN:=50 , IN_WMAX:=800);
	TPV03	:	obj_TPV := (ID:=3, IN_WMIN:=50 , IN_WMAX:=800);
	TPV04	:	obj_TPV := (ID:=4);
	TPV05	:	obj_TPV := (ID:=5);
	TPV06	:	obj_TPV := (ID:=6);

	(* Zigbee temperature probes *)
	ZTHL07	:	obj_ZTHL := (ID:=1, Address:=11); 	(* ZTHL 01 *)
	ZTHL08	:	obj_ZTHL := (ID:=2, Address:=12);	(* ZTHL 02 *)
	ZTHL09	:	obj_ZTHL := (ID:=3, Address:=13);	(* ZTHL 03 *)
	ZTHL10	:	obj_ZTHL := (ID:=4, Address:=14);	(* ZTHL 04 *)
	ZTHL11	:	obj_ZTHL := (ID:=5, Address:=15);	(* ZTHL 05 *)
	ZTHL12	:	obj_ZTHL := (ID:=6, Address:=16);	(* ZTHL 06 *)
	ZTHL13	:	obj_ZTHL := (ID:=7, Address:=17);	(* ZTHL 07 *)

	(** Communication **)
	(* ModBus *)
	MODB01	:	obj_MODBUS		:= (ID:=1, COM:=3, BAUDRATE:=BAUD_19200, RS485:=TRUE);
	MODB02	:	obj_MODBUS_TCP 	:= (ID:=1, IP:='192.168.100.4');

	(* M-Bus *)
	MBUS01	:	obj_MBUS		:= (ID:=1, COM:=2, BAUDRATE:=BAUD_2400);

	(**** SIMULATION ONLY ****)
	(*...*)
END_VAR

(* Global variable list: LON/Module_1/InterfaceBlock_Module_1 *)
VAR_GLOBAL CONSTANT
(******************************************)
(* Automatic generated code, do not edit! *)
(******************************************)
	abSignature_Module_1 : ARRAY[0..15] OF BYTE := 16#0E,16#14,16#D8,16#92,16#C6,16#FC,16#60,16#41,16#91,16#05,16#0D,16#54,16#E3,16#7A,16#DD,16#A3;
	wConfigSize_Module_1 : WORD := 522;
	abInterface_Module_1 : ARRAY[0..130] OF DWORD :=
		16#302841AA, 16#215FDD0C, 16#6041B800, 16#06246830, 16#428B2E71, 16#64B95263, 16#FE000902, 16#2A050140, 
		16#0028C092, 16#037C10FF, 16#6D81026F, 16#0418B0E4, 16#C75C1D07, 16#9CD47157, 16#5A1D2B75, 16#1D531D1E, 
		16#4F0D2658, 16#5AC76C1D, 16#2D5F874A, 16#FE884D09, 16#CE34C958, 16#4CA0345D, 16#856A742A, 16#B26FDD52, 
		16#2BF66959, 16#74C79655, 16#966CD09D, 16#DFE60549, 16#2C48B975, 16#B66DFB76, 16#48BA6ECB, 16#955B162D, 
		16#B7300196, 16#2B35AD5D, 16#65EBC62D, 16#2106DDB9, 16#564CBE30, 16#DDA96F05, 16#AD4B372C, 16#255378CD, 
		16#36ADD181, 16#59D42ACB, 16#9B603585, 16#DDC49858, 16#EA45B329, 16#CD59F616, 16#B50A12E0, 16#56B5BE52, 
		16#8C890100, 16#5AAA1481, 16#B253E154, 16#6C831684, 16#A2ADDCB0, 16#4ABD13A9, 16#950B79D9, 16#4A948694, 
		16#4DBF5E45, 16#CA018948, 16#054C41E5, 16#B86DCB52, 16#2FBEA018, 16#40AAB4D0, 16#A1F866E7, 16#E288A8D1, 
		16#D192DBA2, 16#80E25047, 16#84B4644B, 16#B225A097, 16#59A9F8AC, 16#2D5B376E, 16#7B32E9CE, 16#B7AE3099, 
		16#2D551A30, 16#03F1D236, 16#C96176D0, 16#D94ABD0C, 16#94950479, 16#60B2886A, 16#25C9C990, 16#4CBCB141, 
		16#32D60DA9, 16#6A1D86D9, 16#514404B2, 16#129278D2, 16#09A12969, 16#AB6529E7, 16#90EE2F05, 16#10604094, 
		16#FE031C08, 16#418817F3, 16#84320FB0, 16#238F21C0, 16#6F23C08A, 16#003E98A3, 16#80677304, 16#10728E02, 
		16#0E02FC59, 16#02343A1A, 16#183B223A, 16#804705C0, 16#47864080, 16#47408082, 16#2E208347, 16#A304A014, 
		16#121794C3, 16#81595C58, 16#C785A471, 16#6820171C, 16#7201925C, 16#88CB8581, 16#5D283A17, 16#2378C120, 
		16#1724EF85, 16#0B5F78C0, 16#85687C01, 16#CE17B4F2, 16#814B5FD8, 16#F6856C7D, 16#E8DC173C, 16#6001805F, 
		16#047C0101, 16#97310112, 16#A061674C, 16#20841212, 16#4081A022, 16#A7E890E0, 16#FEC62563, 16#18392858, 
		16#E3A9362C, 16#757477BD, 16#00001088;
END_VAR

(* Global variable list: LON/Module_1/Runtime_Module_1 *)
VAR_GLOBAL
(******************************************)
(* Automatic generated code, do not edit! *)
(******************************************)
	mbxModule_1 : MBX_Full;
	InDataTelegram_Module_1 : ARRAY[0..255] OF BYTE;
	OutDataTelegram_Module_1 : ARRAY[0..511] OF BYTE;

	xInitRunning_Module_1 : BOOL := FALSE;
	unLastLen_mbxModule_1 : UINT;
END_VAR

(* Data type in LON/Enumerations *)
TYPE alarm_type_t :
(
	AL_HEADER := -13,
	AL_FOOTER := -12,
	AL_DEBUG := -11,
	AL_INFO := -10,
	AL_SYSTEM_INFO := -6,
	AL_VALUE_INVALID := -5,
	AL_CONSTANT := -4,
	AL_OFFLINE := -3,
	AL_UNKNOWN := -2,
	AL_NUL := -1,
	AL_NO_CONDITION := 0,
	AL_ALM_CONDITION := 1,
	AL_TOT_SVC_ALM_1 := 2,
	AL_TOT_SVC_ALM_2 := 3,
	AL_TOT_SVC_ALM_3 := 4,
	AL_LOW_LMT_CLR_1 := 5,
	AL_LOW_LMT_CLR_2 := 6,
	AL_HIGH_LMT_CLR_1 := 7,
	AL_HIGH_LMT_CLR_2 := 8,
	AL_LOW_LMT_ALM_1 := 9,
	AL_LOW_LMT_ALM_2 := 10,
	AL_HIGH_LMT_ALM_1 := 11,
	AL_HIGH_LMT_ALM_2 := 12,
	AL_FIR_ALM := 13,
	AL_FIR_PRE_ALM := 14,
	AL_FIR_TRBL := 15,
	AL_FIR_SUPV := 16,
	AL_FIR_TEST_ALM := 17,
	AL_FIR_TEST_PRE_ALM := 18,
	AL_FIR_ENVCOMP_MAX := 19,
	AL_FIR_MONITOR_COND := 20,
	AL_FIR_MAINT_ALERT := 21,
	AL_FATAL_ERROR := 30,
	AL_ERROR := 31,
	AL_WARNING := 32
);
END_TYPE

(* Data type in Logger *)
TYPE en_Logger_ErrLev :
(
	EL_Log			:=0,
	EL_Wrn			:=1,
	EL_Alarm		:=2,
	EL_AlarmStop	:=3
);
END_TYPE

(* Data type in Logger *)
TYPE en_Logger_Status :
(
	S_Logger_UNKNOWN := 0,
	S_Logger_IDLE,
	S_Logger_WAITCONN,
	S_Logger_WAITTX,
	S_Logger_WAITRESP,
	S_Logger_ERROR
);
END_TYPE

(* Data type *)
TYPE en_SYS_Objects :
(
	EO_SYS		:=0,  (* PLC *)
	EO_VPN		:=1,  (* VPN *)
	EO_DOOR		:=2,  (* Door & access control *)

	EO_CAL		:=10, (* Caldaia *)
	EO_CIR		:=11, (* Circolatore *)
	EO_CRON		:=12, (* Crono-termostato *)
	EO_VRD		:=13, (* Valvola miscelatore pannelli *)
	EO_CTL		:=14, (* Contalitri *)
	EO_CTB		:=15, (* Contabilizzatore *)
	EO_TPV		:=16, (* Temperature probes values *)
	EO_PPV		:=17, (* Pressure probes values *)
	EO_PBV		:=18, (* Over-Pressure Alarms *)
	EO_TBV		:=19, (* Over-Temperature Alarms *)
	EO_PMV		:=20, (* Under-Pressure Alarms *)
	EO_GRU		:=21, (* Gruppo termico *)
	EO_PDC		:=22, (* Pompa di calore *)
	EO_SOL		:=23, (* Pannello solare termico *)
	EO_ESOL		:=24, (* Pannello solare fotovoltaico *)
	EO_GAS		:=25, (* Contatore GAS *)
	EO_PORT		:=26, (* Misuratore di portata *)
	EO_FPV		:=27, (* Flow probes values *)
	EO_ANZ		:=28, (* Analizzatore di rete *)
	EO_SCA		:=29, (* Signal Control Alarms *)
	EO_LUX		:=30, (* Base Illumination point *)
	EO_LUXM		:=31, (* Metered Illumination point *)
	EO_PSG		:=32, (* Sensore di passaggio *)
	EO_HVAC		:=33, (* Heating, Ventilating and Air Conditioning *)
	EO_HYGRV	:=34, (* Relative Humidity sensors value *)
	EO_COOV		:=35, (* Carbon Dioxide CO2 sensors value *)
	EO_INV		:=36, (* Inverter *)
	EO_STR		:=37, (* Smart string box *)

	EO_CIRD		:=39, (* Double CIR *)
	EO_ACS		:=40, (* Hot domestic water *)
	EO_FRG		:=41, (* Frigo *)
	EO_THER		:=42, (* Thermostat *)
	EO_CIRM		:=43, (* Modbus CIR *)
	EO_CIRDM	:=44, (* Modbus double CIR *)

	EO_ZGW			:=200,  (* ZigBee - Gateway *)
	EO_ZRM			:=201,	(* ZigBee - Repeater *)
	EO_ZREL			:=202,	(* ZigBee - Actuator rele *)
	EO_ZTHL			:=203,	(* ZigBee - Temperature Sensor *)

	EO_ASGW			:=250,	(* ASi - Gateway *)
	EO_ASCBI		:=251,	(* ASi - Input Board, Ciabatta *)

	EO_LON			:=1000, (* Bus - LON *)
	EO_MODBUS		:=1001, (* Bus - MODBUS *)
	EO_MBUS			:=1002, (* Bus - M-BUS *)
	EO_MODBUS_TCP	:=1003, (* Bus - MODBUS TCP *)

	EO_GENERIC		:=9000, (* Generic dataset *)
	EO_EXPO			:=9001 (* EXPO dataset *)
);
END_TYPE

(* Data type *)
TYPE en_SYS_Status :
(
	S_UNKNOWN  := 0,
	S_STARTUP,
	S_INIT_RTC,
	S_INIT_VAR,
	S_AUTOTEST,
	S_RUNNING,
	S_SHUTDOWN,
	S_HALT
);
END_TYPE

(* Data type in LON/Enumerations *)
TYPE file_request_t :
(
	FR_NUL := -1,
	FR_OPEN_TO_SEND := 0,
	FR_OPEN_TO_RECEIVE := 1,
	FR_CLOSE_FILE := 2,
	FR_CLOSE_DELETE_FILE := 3,
	FR_DIRECTORY_LOOKUP := 4,
	FR_OPEN_TO_SEND_RA := 5,
	FR_OPEN_TO_RECEIVE_RA := 6
);
END_TYPE

(* Data type in LON/Enumerations *)
TYPE file_status_t :
(
	FS_NUL := -1,
	FS_XFER_OK := 0,
	FS_LOOKUP_OK := 1,
	FS_OPEN_FAIL := 2,
	FS_LOOKUP_ERR := 3,
	FS_XFER_UNDERWAY := 4,
	FS_IO_ERR := 5,
	FS_TIMEOUT_ERR := 6,
	FS_WINDOW_ERR := 7,
	FS_AUTH_ERR := 8,
	FS_ACCESS_UNAVAIL := 9,
	FS_SEEK_INVALID := 10,
	FS_SEEK_WAIT := 11
);
END_TYPE

(* Data type in LON/Enumerations *)
TYPE hvac_t :
(
	HVAC_NUL := -1,
	HVAC_AUTO := 0,
	HVAC_HEAT := 1,
	HVAC_MRNG_WRMUP := 2,
	HVAC_COOL := 3,
	HVAC_NIGHT_PURGE := 4,
	HVAC_PRE_COOL := 5,
	HVAC_OFF := 6,
	HVAC_TEST := 7,
	HVAC_EMERG_HEAT := 8,
	HVAC_FAN_ONLY := 9,
	HVAC_FREE_COOL := 10,
	HVAC_ICE := 11,
	HVAC_MAX_HEAT := 12,
	HVAC_ECONOMY := 13,
	HVAC_DEHUMID := 14,
	HVAC_CALIBRATE := 15,
	HVAC_EMERG_COOL := 16,
	HVAC_EMERG_STEAM := 17,
	HVAC_MAX_COOL := 18,
	HVAC_HVC_LOAD := 19,
	HVAC_NO_LOAD := 20
);
END_TYPE

(* Data type in LON/Enumerations *)
TYPE object_request_t :
(
	RQ_NUL := -1,
	RQ_NORMAL := 0,
	RQ_DISABLED := 1,
	RQ_UPDATE_STATUS := 2,
	RQ_SELF_TEST := 3,
	RQ_UPDATE_ALARM := 4,
	RQ_REPORT_MASK := 5,
	RQ_OVERRIDE := 6,
	RQ_ENABLE := 7,
	RQ_RMV_OVERRIDE := 8,
	RQ_CLEAR_STATUS := 9,
	RQ_CLEAR_ALARM := 10,
	RQ_ALARM_NOTIFY_ENABLED := 11,
	RQ_ALARM_NOTIFY_DISABLED := 12,
	RQ_MANUAL_CTRL := 13,
	RQ_REMOTE_CTRL := 14,
	RQ_PROGRAM := 15,
	RQ_CLEAR_RESET := 16,
	RQ_RESET := 17,
	RQ_CLEAR_LOG := 18,
	RQ_LOAD_PROGRAM := 19,
	RQ_RUN_PROGRAM := 20,
	RQ_HALT_PROGRAM := 21,
	RQ_RESTART_PROGRAM := 22,
	RQ_UNLOAD_PROGRAM := 23,
	RQ_STEP_PROGRAM := 24
);
END_TYPE

(* Data type in LON/Enumerations *)
TYPE priority_level_t :
(
	PR_NUL := -1,
	PR_LEVEL_0 := 0,
	PR_LEVEL_1 := 1,
	PR_LEVEL_2 := 2,
	PR_LEVEL_3 := 3,
	PR_1 := 4,
	PR_2 := 5,
	PR_3 := 6,
	PR_4 := 7,
	PR_6 := 8,
	PR_8 := 9,
	PR_10 := 10,
	PR_16 := 11
);
END_TYPE

(* Data type in Plant_Objects *)
TYPE typ_Clima : (* CURVA CLIMATICA *)
STRUCT
	InitOK:		BOOL;
	Points: 	ARRAY [0..10] OF POINT;
END_STRUCT
END_TYPE

(* Data type in Plant_Objects *)
TYPE typ_Cron_Calendar :
STRUCT
	Profile		: ARRAY[0..384] OF BYTE;
END_STRUCT
END_TYPE

(* Data type in Plant_Objects *)
TYPE typ_Cron_Jolly :
STRUCT
	Start		: DT;
	End			: DT;
	Temp		: WORD;
	Flags		: WORD; (* B0:Enabled B1..B15:Unused *)
END_STRUCT
END_TYPE

(* Data type in Plant_Objects *)
TYPE typ_Cron_Profile :
STRUCT
	Flags		: WORD;
	Setpoint	: ARRAY [0..95] OF WORD;
END_STRUCT
END_TYPE

(* Data type in Logger *)
TYPE typ_Logger :
STRUCT
	Status		: en_Logger_Status;

	SendReq		: BOOL;
	SendIdx		: DWORD;
	SendData	: ARRAY [0..MAX_SEND_TCP_CLIENT] OF BYTE;
	SendLen		: DINT;

	TData		: ARRAY [0..MAX_SEND_TCP_CLIENT] OF BYTE;
	TLen		: DINT;

	LastIdxPos	: DWORD;

	(* Temporary variables used by objects *)
	s1			: STRING(256);
	i1			: WORD;

END_STRUCT
END_TYPE

(* Data type in Plant_Objects *)
TYPE typ_MODBUS_ABB_DMTME72 :
STRUCT
	V_3P		: DWORD; (* V *)
	V_L1N		: DWORD;
	V_L2N		: DWORD;
	V_L3N		: DWORD;
	V_L1L2		: DWORD;
	V_L2L3		: DWORD;
	V_L3L1		: DWORD;
	I_3P		: DWORD; (* 10^-3 A *)
	I_L1		: DWORD;
	I_L2		: DWORD;
	I_L3		: DWORD;
	PF_3P		: DINT;	 (* 10^-3 *)
	PF_L1		: DINT;
	PF_L2		: DINT;
	PF_L3		: DINT;
	COS_3P		: DINT;  (*NO!*)
	COS_L1		: DINT;
	COS_L2		: DINT;
	COS_L3		: DINT;
	VA_3P		: DWORD; (* VA *)(*NO!*)
	VA_L1		: DWORD;
	VA_L2		: DWORD;
	VA_L3		: DWORD;
	P_3P		: DWORD; (* W *)
	P_L1		: DWORD;
	P_L2		: DWORD;
	P_L3		: DWORD;
	Q_3P		: DWORD; (* VAr *)
	Q_L1		: DWORD;
	Q_L2		: DWORD;
	Q_L3		: DWORD;

	WH_3P		: DWORD; (* 10^-1 kWh *)
	VARH_3P		: DWORD; (* 10^-1 kVArh *)
	FREQ		: DWORD; (* 10^-3 Hz *)

	I_L1_Max	: DWORD;
	I_L2_Max	: DWORD;
	I_L3_Max	: DWORD;
	P_3P_Max	: DWORD;
	Q_3P_Max	: DWORD;
	P_3P_Avg15m	: DWORD;

END_STRUCT
END_TYPE

(* Data type in Plant_Objects *)
TYPE typ_MODBUS_CIR :
STRUCT
	PumpStatus		:	WORD;
	PumpFault		:	BOOL;
	PumpBoardTemp	:	INT;	(* Electonic board temperature  [°C] *)
	PumpVoltage		:	WORD;	(* Input voltage rms [V] *)
	PumpCurrent		:	WORD;	(* Output current [E-3 A]	*)
	PumpRPM			:	WORD;	(* Round per minute [rpm] *)
	PumpPower		:	WORD;	(* Power [W] *)
	PumpOpTime		:	DWORD;	(* Pump operating time [h] *)
	PumpHead		:	WORD;	(* [E-1 m] *)
	PumpFlow		:	WORD;	(* Extimated flow [E-1 m3/h] *)
	PumpLiqTemp		:	WORD;	(* Liquid temperature [°C] *)
	PumpAlarm		:	ARRAY [0..14] OF WORD;

END_STRUCT
END_TYPE

(* Data type in Plant_Objects *)
TYPE typ_MODBUS_ELGAS_MINIELCOR :
STRUCT
	Vb			: ARRAY [0..3] OF WORD;	(* m^3 *)
	Vm			: DWORD;				(* m^3 *)
	P			: REAL;					(* bar *)
	T			: REAL;					(* °C *)
	C			: REAL;
	Vbs			: ARRAY [0..3] OF WORD;	(* m^3 *)
	Vb_d_d		: ARRAY [0..3] OF WORD;	(* m^3 *)
	Vb_d_m		: ARRAY [0..3] OF WORD;	(* m^3 *)
	Vm_d_d		: DWORD;				(* m^3 *)
	Q			: REAL;					(* m^3/h *)
	Qb			: REAL;					(* m^3/h *)

	BC_EVC		: REAL;			(* % *)
	BV_EVC		: REAL;			(* V *)
	D_Err		: WORD;			(* 0:OK, 1:FAIL *)
	Status		: DWORD;		(* Status bits *)

END_STRUCT
END_TYPE

(* Data type in Plant_Objects *)
TYPE typ_MODBUS_FRER_IQ96U2 :
STRUCT
	V_L1N		: DWORD; (* 10^-3 V *)
	V_L2N		: DWORD;
	V_L3N		: DWORD;
	V_L1L2		: DWORD;
	V_L2L3		: DWORD;
	V_L3L1		: DWORD;
	I_L1		: DWORD; (* 10^-3 I *)
	I_L2		: DWORD;
	I_L3		: DWORD;
	FREQ		: DWORD; (* 10^-3 Hz *)
	P_3P		: DWORD; (* W *)
	Q_3P		: DWORD; (* VAr *)
	PF_3P		: DINT;	 (* 10^-3 *)
	WH_3P		: DWORD; (* Wh *)
	VARH_3P		: DWORD; (* VArh *)
	MULT		: DWORD;

	WH_3P_NEG	: DWORD; (* Wh *)
	VARH_3P_NEG : DWORD; (* VArh *)
	S_3P		: DWORD; (* VA *)

	PF_L1		: DWORD; (* 10^-3 *)
	PF_L2		: DWORD; (* 10^-3 *)
	PF_L3		: DWORD; (* 10^-3 *)

	P_3P_Max	: DWORD;
	P_3P_Avg15m	: DWORD;
	I_L1_Max	: DWORD;
	I_L2_Max	: DWORD;
	I_L3_Max	: DWORD;
	I_L1_Avg15m	: DWORD;
	I_L2_Avg15m	: DWORD;
	I_L3_Avg15m	: DWORD;

END_STRUCT
END_TYPE

(* Data type in Plant_Objects *)
TYPE typ_MODBUS_VAR : (* Gestione parametri MODBUS *)
STRUCT
	SlaveAddress	: BYTE;
	FunCode			: BYTE;
	FunAddress		: WORD;
	Refresh_Time	: BYTE; (* 0:No refresh x:Refresh in seconds *)
	Refresh_Cnt		: BYTE; (* INTERNAL *)
	Variable		: POINTER TO WORD;
	Variable_Size	: BYTE;
	Variable_Mirror : WORD; (* INTERNAL [Force refresh on read variables when <>0] *)
END_STRUCT
END_TYPE

(* Data type *)
TYPE typ_SYS :
STRUCT
	Status			: en_SYS_Status;
	Warning			: BOOL;
	Alarm			: BOOL;
	AlarmStop		: BOOL;

	Time_LogString	: STRING;
	Time_Year		: WORD;
	Time_Month		: BYTE;
	Time_Day		: BYTE;
	Time_Hour		: BYTE;
	Time_Minute		: BYTE;

	Time_CT_DT		: DT;
	Time_CT_Day		: WORD;
	Time_CT_Quarter	: BYTE;

	LastLogs_Idx	: BYTE;
	LastLogs_Dat	: ARRAY[0..5] OF STRING;
	LastLogs_Msg	: ARRAY[0..5] OF STRING;

END_STRUCT
END_TYPE

(* Data type in Plant_Objects *)
TYPE typ_VisuStrutturaMbus :
STRUCT

	sdNodoPresente: STRING(16);
	sdEnergia: STRING(16);
	sdPotenza: STRING(16);
	sdVolume: STRING(16);
	sdFlow: STRING(16);
	sdTempIngresso: STRING(8);
	sdTempaUscita: STRING(8);
	sdTempDelta: STRING(8);

END_STRUCT
END_TYPE

(* Data type in LON/NetworkVariables *)
TYPE typSnvtAlarm : 
STRUCT
	abLocation : ARRAY[0..5] OF BYTE;
	wObjectId : WORD;
	bAlarmType : BYTE (* enum type alarm_type_t *);
	bPriorityLevel : BYTE (* enum type priority_level_t *);
	wIndexToSnvt : WORD;
	abValue : ARRAY[0..3] OF BYTE;
	wYear : WORD;
	bMonth : BYTE;
	bDay : BYTE;
	bHour : BYTE;
	bMinute : BYTE;
	bSecond : BYTE;
	wMillisecond : WORD;
	abAlarmLimit : ARRAY[0..3] OF BYTE;
	bStatusInformation : BYTE; (* bit allocation of bStatusInformation:
	bit 0: NVI update counter LSB
	bit 1: NVI update counter
	bit 2: NVI update counter
	bit 3: NVI update counter MSB
	bit 4: timeout for NVI occurs (MaxRcvTime expired)
	bit 5: reserved
	bit 6: reserved
	bit 7: force NVO update *)
	bInternalUseOnly : BYTE; (* Do not use this byte in your application! *)
END_STRUCT
END_TYPE

(* Data type in LON/NetworkVariables *)
TYPE typSnvtFilePos : 
STRUCT
	diRwPtr : DINT;
	wRwLength : WORD;
	bStatusInformation : BYTE; (* bit allocation of bStatusInformation:
	bit 0: NVI update counter LSB
	bit 1: NVI update counter
	bit 2: NVI update counter
	bit 3: NVI update counter MSB
	bit 4: timeout for NVI occurs (MaxRcvTime expired)
	bit 5: reserved
	bit 6: reserved
	bit 7: force NVO update *)
	bInternalUseOnly : BYTE; (* Do not use this byte in your application! *)
END_STRUCT
END_TYPE

(* Data type in LON/NetworkVariables *)
TYPE typSnvtFileReq : 
STRUCT
	bRequest : BYTE (* enum type file_request_t *);
	wIndex : WORD;
	wReceiveTimeout : WORD;
	abDestAddress : ARRAY[0..4] OF BYTE (* union declaration *);
	bAuthOn : BYTE;
	bPrioOn : BYTE;
	bStatusInformation : BYTE; (* bit allocation of bStatusInformation:
	bit 0: NVI update counter LSB
	bit 1: NVI update counter
	bit 2: NVI update counter
	bit 3: NVI update counter MSB
	bit 4: timeout for NVI occurs (MaxRcvTime expired)
	bit 5: reserved
	bit 6: reserved
	bit 7: force NVO update *)
	bInternalUseOnly : BYTE; (* Do not use this byte in your application! *)
END_STRUCT
END_TYPE

(* Data type in LON/NetworkVariables *)
TYPE typSnvtFileStatus : 
STRUCT
	bStatus : BYTE (* enum type file_status_t *);
	wNumberOfFiles : WORD;
	wSelectedFile : WORD;
	abAdr : ARRAY[0..21] OF BYTE (* union declaration *);
	bStatusInformation : BYTE; (* bit allocation of bStatusInformation:
	bit 0: NVI update counter LSB
	bit 1: NVI update counter
	bit 2: NVI update counter
	bit 3: NVI update counter MSB
	bit 4: timeout for NVI occurs (MaxRcvTime expired)
	bit 5: reserved
	bit 6: reserved
	bit 7: force NVO update *)
	bInternalUseOnly : BYTE; (* Do not use this byte in your application! *)
END_STRUCT
END_TYPE

(* Data type in LON/NetworkVariables *)
TYPE typSnvtHvacMode : 
STRUCT
	bSnvtHvacMode : BYTE (* enum type hvac_t *);
	bStatusInformation : BYTE; (* bit allocation of bStatusInformation:
	bit 0: NVI update counter LSB
	bit 1: NVI update counter
	bit 2: NVI update counter
	bit 3: NVI update counter MSB
	bit 4: timeout for NVI occurs (MaxRcvTime expired)
	bit 5: reserved
	bit 6: reserved
	bit 7: force NVO update *)
	bInternalUseOnly : BYTE; (* Do not use this byte in your application! *)
END_STRUCT
END_TYPE

(* Data type in LON/NetworkVariables *)
TYPE typSnvtObjRequest : 
STRUCT
	wObjectId : WORD;
	bObjectRequest : BYTE (* enum type object_request_t *);
	bStatusInformation : BYTE; (* bit allocation of bStatusInformation:
	bit 0: NVI update counter LSB
	bit 1: NVI update counter
	bit 2: NVI update counter
	bit 3: NVI update counter MSB
	bit 4: timeout for NVI occurs (MaxRcvTime expired)
	bit 5: reserved
	bit 6: reserved
	bit 7: force NVO update *)
	bInternalUseOnly : BYTE; (* Do not use this byte in your application! *)
END_STRUCT
END_TYPE

(* Data type in LON/NetworkVariables *)
TYPE typSnvtObjStatus : 
STRUCT
	wObjectId : WORD;
	bBitfieldByteOffset2 : BYTE (* bit field *);
	bBitfieldByteOffset3 : BYTE (* bit field *);
	bBitfieldByteOffset4 : BYTE (* bit field *);
	bBitfieldByteOffset5 : BYTE (* bit field *);
	bStatusInformation : BYTE; (* bit allocation of bStatusInformation:
	bit 0: NVI update counter LSB
	bit 1: NVI update counter
	bit 2: NVI update counter
	bit 3: NVI update counter MSB
	bit 4: timeout for NVI occurs (MaxRcvTime expired)
	bit 5: reserved
	bit 6: reserved
	bit 7: force NVO update *)
	bInternalUseOnly : BYTE; (* Do not use this byte in your application! *)
END_STRUCT
END_TYPE

(* Data type in LON/NetworkVariables *)
TYPE typSnvtState : 
STRUCT
	bBitfieldByteOffset0 : BYTE (* bit field *);
	bBitfieldByteOffset1 : BYTE (* bit field *);
	bStatusInformation : BYTE; (* bit allocation of bStatusInformation:
	bit 0: NVI update counter LSB
	bit 1: NVI update counter
	bit 2: NVI update counter
	bit 3: NVI update counter MSB
	bit 4: timeout for NVI occurs (MaxRcvTime expired)
	bit 5: reserved
	bit 6: reserved
	bit 7: force NVO update *)
	bInternalUseOnly : BYTE; (* Do not use this byte in your application! *)
END_STRUCT
END_TYPE

(* Data type in LON/NetworkVariables *)
TYPE typSnvtSwitch : 
STRUCT
	bValue : BYTE;
	siState : SINT;
	bStatusInformation : BYTE; (* bit allocation of bStatusInformation:
	bit 0: NVI update counter LSB
	bit 1: NVI update counter
	bit 2: NVI update counter
	bit 3: NVI update counter MSB
	bit 4: timeout for NVI occurs (MaxRcvTime expired)
	bit 5: reserved
	bit 6: reserved
	bit 7: force NVO update *)
	bInternalUseOnly : BYTE; (* Do not use this byte in your application! *)
END_STRUCT
END_TYPE

(* Data type in LON/NetworkVariables *)
TYPE typSnvtTempP : 
STRUCT
	iSnvtTempP : INT;
	bStatusInformation : BYTE; (* bit allocation of bStatusInformation:
	bit 0: NVI update counter LSB
	bit 1: NVI update counter
	bit 2: NVI update counter
	bit 3: NVI update counter MSB
	bit 4: timeout for NVI occurs (MaxRcvTime expired)
	bit 5: reserved
	bit 6: reserved
	bit 7: force NVO update *)
	bInternalUseOnly : BYTE; (* Do not use this byte in your application! *)
END_STRUCT
END_TYPE

(* Data type in LON/NetworkVariables *)
TYPE typSnvtTimeStamp : 
STRUCT
	iYear : INT;
	bMonth : BYTE;
	bDay : BYTE;
	bHour : BYTE;
	bMinute : BYTE;
	bSecond : BYTE;
	bStatusInformation : BYTE; (* bit allocation of bStatusInformation:
	bit 0: NVI update counter LSB
	bit 1: NVI update counter
	bit 2: NVI update counter
	bit 3: NVI update counter MSB
	bit 4: timeout for NVI occurs (MaxRcvTime expired)
	bit 5: reserved
	bit 6: reserved
	bit 7: force NVO update *)
	bInternalUseOnly : BYTE; (* Do not use this byte in your application! *)
END_STRUCT
END_TYPE

(* POU PLC_PRG, ST *)
PROGRAM PLC_PRG
VAR
	Timer1: TON; (* Fast controls tick *)
	Timer2: TON; (* Plant control tick *)
	Timer3: TON; (* Logger timer *)

	T_CIRD01	:	INT;
	T_CIRD02	:	INT;
	T_CIRD03	:	INT;
	T_CIRD04	:	INT;
	T_CIRD05	:	INT;
	T_CIRD06	:	INT;

	T_CIR03		:	INT;

	T_VRD01		:	INT;
	T_VRD02		:	INT;
	T_VRD03		:	INT;

	SecCircuitLogic	:	BOOL;	(* Secondary circuit request: LOGICAL ON/OFF *)
	SecCircuitReal	:	BOOL;	(* Secondart circuit request: REAL ON/OFF	 *)
	Gain: INT;
	test: BOOL;
	Gain1: REAL;
	Gain2: REAL;
	Gain3: REAL;

	ErroreAcqua: INT;


	StartCAL_Antigelo: RS;
	fAntigelo		:FLT_TAP;  (* Sgnalazione LOG Antigelo  *)




END_VAR
(******************************************************************************
 ****                           MAIN TASK CODE                             ****
 ******************************************************************************

	Network setup:
		IP  = 192.168.100.2 | MSK = 255.255.255.0
		GW	= 192.168.100.1 | DNS = 192.168.100.1
		SNTP = 193.204.114.232 (3600s) ==> 192.168.100.3

*)

(*==============================*)
(*===== Main status machine ====*)
(*==============================*)
Main_Stm();

(*==============================*)
(*== Running cycle operations ==*)
(*==============================*)
IF SYS.Status>S_INIT_VAR THEN
	(* Execute cycle processes *)
	(* Update LON output variables (needs to be here to obtain only one refresh) *)
	CAL01.Heartbeat( CLIM:=CAL01_Clima );
	CAL02.Heartbeat( CLIM:=CAL02_Clima );
	(* Execute LON process *)
	Module_1_PRG();

	(* Count water pulses *)
	CTL01(CTL_ST:=CTL01_ST, COUNT:=Ctl01_Counter);
	CTL02(CTL_ST:=CTL02_ST, COUNT:=Ctl02_Counter);

	(* ModBus *)
	MODB01();

	CIR01(ModBus:=MODB01, Pump_AL:=NOT CIR01_AL, Pump_AUTO:=NOT CIR01_AUTO, OnOff:=SecCircuitReal);
	CIR02(ModBus:=MODB01, Pump_AL:=NOT CIR02_AL, Pump_AUTO:=NOT CIR02_AUTO, CTRL_Run=>CAL02.Run);

	CIRD01(ModBus:=MODB01, PumpA_AL:=NOT CIRD01_A_AL, PumpB_AL:=NOT CIRD01_B_AL, PumpA_AUTO:=NOT CIRD01_A_AUTO, PumpB_AUTO:=NOT CIRD01_B_AUTO);
	CIRD02(ModBus:=MODB01, PumpA_AL:=NOT CIRD02_A_AL, PumpB_AL:=NOT CIRD02_B_AL, PumpA_AUTO:=NOT CIRD02_A_AUTO, PumpB_AUTO:=NOT CIRD02_B_AUTO);
	CIRD03(ModBus:=MODB01, PumpA_AL:=NOT CIRD03_A_AL, PumpB_AL:=NOT CIRD03_B_AL, PumpA_AUTO:=NOT CIRD03_A_AUTO, PumpB_AUTO:=NOT CIRD03_B_AUTO);
	CIRD04(ModBus:=MODB01, PumpA_AL:=NOT CIRD04_A_AL, PumpB_AL:=NOT CIRD04_B_AL, PumpA_AUTO:=NOT CIRD04_A_AUTO, PumpB_AUTO:=NOT CIRD04_B_AUTO);
	CIRD05(ModBus:=MODB01, PumpA_AL:=NOT CIRD05_A_AL, PumpB_AL:=NOT CIRD05_B_AL, PumpA_AUTO:=NOT CIRD05_A_AUTO, PumpB_AUTO:=NOT CIRD05_B_AUTO);

NodoDaInterrogare:=LIMIT(1,NodoDaInterrogare,13);
IF NodoDaInterrogare>12 THEN NodoDaInterrogare:=1;END_IF;


	(* Pump *)
	CIR03(Pump_AL:=NOT CIR03_AL, Pump_ST:=CIR03_ST, Pump_AUTO:=NOT CIR03_AUTO, CIR_EN=>CIR03_EN);

	(* Double pumps *)
	CIRD06(PumpA_AL:=NOT CIRD06_A_AL, PumpB_AL:=NOT CIRD06_B_AL, PumpA_ST:=CIRD06_A_ST, PumpB_ST:=CIRD06_B_ST,
			   PumpA_AUTO:=NOT CIRD06_A_AUTO, PumpB_AUTO:=NOT CIRD06_B_AUTO );




	(* TCP ModBus *)
	MODB02();

	ZTHL07(MODBUS:=MODB02);
	ZTHL08(MODBUS:=MODB02);
	ZTHL09(MODBUS:=MODB02);
	ZTHL10(MODBUS:=MODB02);
	ZTHL11(MODBUS:=MODB02);
	ZTHL12(MODBUS:=MODB02);
	ZTHL13(MODBUS:=MODB02);

	(* M-Bus *)
	MBUS01();

	CTB01(MBUS:=MBUS01);

END_IF

(*==============================*)
(*== System cycle operations ===*)
(*==============================*)
(* Execute TCP processes *)
Logger_Proc();
Remote_Proc();
(* Update user led *)
USRLED_Update();
(* Execute Cron Editor commands *)
CronEd();

(* Environment temperature *)
IF NOT TPV01.ERR THEN T_AMB := S01;
ELSE T_AMB := Plant_DefaultTAmb;
END_IF


(**** SIMULATION ONLY ****)
(*...*)
END_PROGRAM
ACTION Main_Stm:
CASE Sys.Status OF

	S_STARTUP:
		Sys.Status:=S_INIT_RTC;

	S_INIT_RTC:
		(* Check RTC and update from network *)
		RTC_Update();
		(* Check time *)
		IF Sys.Time_Year>2000 THEN
			Sys.Status:=S_INIT_VAR;
		END_IF

	S_INIT_VAR:
		LogEv(EL_Wrn,EO_SYS,0,1,CONCAT('System_startup_v',WORD_TO_STRING(Plant_SW_VER)));
		Sys.Status:=S_RUNNING;

	S_RUNNING:
		Timer1(IN:=NOT Timer1.Q,PT:=T#50ms);
		IF Timer1.Q THEN
			(* Update meters *)

			(* Update system checks *)
			SYS_Proc();
		END_IF

		Timer2(IN:=NOT Timer2.Q,PT:=T#500ms);
		IF Timer2.Q THEN
			(* Read current date/time *)
			RTC_Update();


			(* Temperature *)
			T_CIRD01 := ZTHL07.OUT_TEMP;   	(* ZTHL01 Salone Materna Ventilatore *)
			T_CIRD02 := ZTHL08.OUT_TEMP;	(* ZTHL02 PT Materna  *)
			T_CIRD06 := ZTHL09.OUT_TEMP;	(* ZTHL03 Palestra  1°P Elementare *)
			T_CIRD03 := ZTHL11.OUT_TEMP;	(* ZTHL05 Aule  PT Elementare *)
			T_CIRD04 := ZTHL12.OUT_TEMP;	(* ZTHL06 Mensa Elementare *)
			T_CIRD05 := ZTHL13.OUT_TEMP;	(* ZTHL07 Uffici Seminterrato *)

			T_CIR03 := ZTHL10.OUT_TEMP;	 	(* ZTHL04 Aule  1°P Elementare *)


	(* Gestione Ciclo antigelo : in questo impianto il ciclo antigelo è gestito coi crono ambiente *)

			StartCAL_Antigelo(	SET:=(SogliaMinStartAntigelo>TPV03.AVG),
								RESET1:= (TPV03.AVG>SogliaMinStopAntigelo) OR NOT BitAbilitaAntigelo
							);

			fAntigelo(IN:=StartCAL_Antigelo.Q1);
			IF fAntigelo.EVH THEN
				LogEv(EL_Log,EO_SYS,0,11,'Ciclo_Antigelo_Attivato');
			END_IF
			IF fAntigelo.EVL THEN
				LogEv(EL_Log,EO_SYS,0,12,'Ciclo_Antigelo_Disattivato');
			END_IF




			(* Thermostats *)
			(* CIRDM01 *)
			THER01(Temperature:=T_CIRD01);(* AntifreezeForce=>CIRD01.CIR_RUN_REQ);*)
			CIRD01.OnOff:=SEL(ZTHL07.ERR,THER01.Run,THER01.RunCrono) OR StartCAL_Antigelo.Q1; (* Salone Materna Ventilatore *)

			(* CIRDM02 *)
			THER02(Temperature:=T_CIRD02);(*, AntifreezeForce=>CIRD02.CIR_RUN_REQ);*)
			CIRD02.OnOff:=SEL(ZTHL08.ERR,THER02.Run,THER02.RunCrono) OR StartCAL_Antigelo.Q1;


			(* CIRDM03 *)
			THER03(Temperature:=T_CIRD03);(*, AntifreezeForce=>CIRD03.CIR_RUN_REQ);*)
			CIRD03.OnOff:=SEL(ZTHL09.ERR,THER03.Run,THER03.RunCrono) OR StartCAL_Antigelo.Q1;

			(* CIRDM04 *)
			THER04(Temperature:=T_CIRD04);(*, AntifreezeForce=>CIRD04.CIR_RUN_REQ);*)
			CIRD04.OnOff:=SEL(ZTHL12.ERR,THER04.Run,THER04.RunCrono) OR StartCAL_Antigelo.Q1;

			(* CIRDM05 *)
			THER05(Temperature:=T_CIRD05);(*, AntifreezeForce=>CIRD05.CIR_RUN_REQ);*)
			CIRD05.OnOff:=SEL(ZTHL11.ERR,THER05.Run,THER05.RunCrono) OR StartCAL_Antigelo.Q1;

			(* CIRD01 *)
			THER06(Temperature:=T_CIRD06);(*, AntifreezeForce=>CIRD06.CIR_RUN_REQ);*)
			CIRD06.OnOff:=SEL(ZTHL13.ERR,THER06.Run,THER06.RunCrono) OR StartCAL_Antigelo.Q1;

			(* CIRD01 *)
			THER07(Temperature:=T_CIR03);
			CIR03.OnOff:=SEL(ZTHL07.ERR,THER07.Run,THER07.RunCrono) OR StartCAL_Antigelo.Q1;



		(* questa modifica si è resa necessaria perchè in relatà il cird06 ha una pompa che non c'è *)
			CIRD06_A_EN:=CIRD06.PumpA_En OR CIRD06.PumpB_En;
			CIRD06_B_EN:=CIRD06.PumpA_En OR CIRD06.PumpB_En;


			THER250();


			(* Probes *)
			TPV01(IN:=S01);
			TPV02(IN:=S02);
			TPV03(IN:=S03);
			TPV04(IN:=S04);
			TPV05(IN:=S05);
			TPV06(IN:=S06);

			T_VRD01 := SEL(TPV04.ERR,TPV04.IN,Plant_VRD_TDefault);
			T_VRD02 := SEL(TPV05.ERR,TPV05.IN,Plant_VRD_TDefault);
			T_VRD03 := SEL(TPV06.ERR,TPV06.IN,Plant_VRD_TDefault);

			(* Valves *)
			VRD01(RUN:=CIRD01.Run,OffsetBoost:=THER250.SetPoint, CLIM:=VRD01_Clima, TEMP:=T_VRD01, STATUS:=VRD01_ST, OUT_CL=>VRD01_CL, OUT_OP=>VRD01_OP);
			VRD02(RUN:=CIRD02.Run,OffsetBoost:=THER250.SetPoint, CLIM:=VRD02_Clima, TEMP:=T_VRD02, STATUS:=VRD02_ST, OUT_CL=>VRD02_CL, OUT_OP=>VRD02_OP);
			VRD03(RUN:=(CIR03.Run OR CIRD03.Run OR CIRD04.Run OR CIRD05.Run),OffsetBoost:=THER250.SetPoint, CLIM:=VRD03_Clima, TEMP:=T_VRD03, STATUS:=VRD03_ST, OUT_CL=>VRD03_CL, OUT_OP=>VRD03_OP);


			(* Calcolo l'errore dell'acqua mandata e ritorno in modo da controllare la velocità delle pompe di mandata *)
			ErroreAcqua:=STRING_TO_INT(CTB01.M1.utFTemp.Value)-STRING_TO_INT(CTB01.M1.utRTemp.Value);

			Gain1:=INT_TO_REAL(PercVelMax-PercVelMin)/INT_TO_REAL(ErroreTempMax-ErroreTempMin);
			Gain2:=Gain1*INT_TO_REAL(ErroreAcqua-ErroreTempMin);
			Gain3:=Gain2 + INT_TO_REAL(PercVelMin);
			Gain:=LIMIT(REAL_TO_INT(Gain3),PercVelMin,PercVelMax);

			CIR01.VelocitaRichiesta:=Gain;
			CIR02.VelocitaRichiesta:=Gain;


			(* Secondary circuit heat request *)
			SecCircuitLogic := CIRD01.Ctrl_Run OR CIRD02.Ctrl_Run OR CIRD03.Ctrl_Run OR CIRD04.Ctrl_Run OR CIRD05.Ctrl_Run OR CIRD06.Ctrl_Run OR CIR03.Ctrl_Run;
			SecCircuitReal	:= CIRD01.Run OR CIRD02.Run OR CIRD03.Run OR CIRD04.Run OR CIRD05.Run OR CIRD06.Run OR CIR03.Run;

			(* No secondary circuit heat request -->> Switch off immediatly CAL
			   Secondary circuit heat request -->> First switch on primary pump CIR01, when enabled switch on CAL *)

			(* Comando Ciroclatore Primario *)
			CIR01.OnOff := SEL(SecCircuitLogic,FALSE,TRUE) AND SYS.AlarmStop=FALSE;
			CAL01.Run := SEL(SecCircuitLogic,FALSE,CIR01.Run) AND SYS.AlarmStop=FALSE;

			(* Boilers cascade *)
			(* ATTENZIONE il valore che restituisce il LON è a 2 decimali *)
			CAS01(RUN_Primary:=SEL(SecCircuitLogic,FALSE,CIR01.Run) AND SYS.AlarmStop=FALSE, SetTemp:=CAL01.Curve_Temp , ReadTemp:=S02 + OffsetSetPointManuale , OUT_Secondary=>CIR02.OnOff);

			(* Scrivo il setpoint in funzione della curva cliamatica più alta *)

			CAL01.SetPointManuale:=CAL01.Curve_Temp - OffsetSetPointManuale;
			CAL01.SetPointManuale:=MAX(CAL01.SetPointManuale,SEL(VRD01.RUN,0,VRD01.Ctrl_SetPoint));
			CAL01.SetPointManuale:=MAX(CAL01.SetPointManuale,SEL(VRD02.RUN,0,VRD02.Ctrl_SetPoint));
			CAL01.SetPointManuale:=MAX(CAL01.SetPointManuale,SEL(VRD03.RUN,0,VRD03.Ctrl_SetPoint));


			CAL02.SetPointManuale:=CAL01.SetPointManuale;

			CAL01(CLIM:=CAL01_Clima,AbilitaSetPointManuale:=TRUE);
			CAL02(CLIM:=CAL01_Clima,AbilitaSetPointManuale:=TRUE);


			Lamp( Allarme:=	CAL01.Status_Log=2 OR
							CAL02.Status_Log=2 OR
 							CTL01.Status_Log=2 OR
							CTL02.Status_Log=2 OR
							CTB01.Status_Log=2 OR
							THER01.Status_Log=2 OR
							THER02.Status_Log=2 OR
							THER03.Status_Log=2 OR
							THER04.Status_Log=2 OR
							THER05.Status_Log=2 OR
							THER06.Status_Log=2 OR
							THER07.Status_Log=2 OR
							THER250.Status_Log=2 OR
							VRD01.Status_Log=2 OR
							VRD02.Status_Log=2 OR
							VRD03.Status_Log=2 OR
							CIR01.Status_Log=2 OR
  						  	CIR02.Status_Log=2 OR
  						  	CIR03.Status_Log=2 OR
   						  	CIRD01.Status_Log=2 OR
 						  	CIRD02.Status_Log=2 OR
						  	CIRD03.Status_Log=2 OR
						  	CIRD04.Status_Log=2 OR
						  	CIRD05.Status_Log=2 OR
						  	CIRD06.Status_Log=2 OR
							TPV01.Status_Log=2 OR
							TPV02.Status_Log=2 OR
							TPV03.Status_Log=2 OR
							TPV04.Status_Log=2 OR
							TPV05.Status_Log=2 OR
							TPV06.Status_Log=2 OR
							ZTHL07.Status_Log=2 OR
							ZTHL08.Status_Log=2 OR
							ZTHL09.Status_Log=2 OR
							ZTHL10.Status_Log=2 OR
							ZTHL11.Status_Log=2 OR
							ZTHL12.Status_Log=2 OR
							ZTHL13.Status_Log=2 OR
							MODB01.Status_Log=2 OR
							MODB02.Status_Log=2 OR
							MBUS01.Status_Log=2,
							Warning:=CAL01.Status_Log=1 OR
							CAL02.Status_Log=1 OR
 							CTL01.Status_Log=1 OR
							CTL02.Status_Log=1 OR
							CTB01.Status_Log=1 OR
							THER01.Status_Log=1 OR
							THER02.Status_Log=1 OR
							THER03.Status_Log=1 OR
							THER04.Status_Log=1 OR
							THER05.Status_Log=1 OR
							THER06.Status_Log=1 OR
							THER07.Status_Log=1 OR
							THER250.Status_Log=1 OR
							VRD01.Status_Log=1 OR
							VRD02.Status_Log=1 OR
							VRD03.Status_Log=1 OR
							CIR01.Status_Log=1 OR
  						  	CIR02.Status_Log=1 OR
  						  	CIR03.Status_Log=1 OR
   						  	CIRD01.Status_Log=1 OR
 						  	CIRD02.Status_Log=1 OR
						  	CIRD03.Status_Log=1 OR
						  	CIRD04.Status_Log=1 OR
						  	CIRD05.Status_Log=1 OR
						  	CIRD06.Status_Log=1 OR
							TPV01.Status_Log=1 OR
							TPV02.Status_Log=1 OR
							TPV03.Status_Log=1 OR
							TPV04.Status_Log=1 OR
							TPV05.Status_Log=1 OR
							TPV06.Status_Log=1 OR
							ZTHL07.Status_Log=1 OR
							ZTHL08.Status_Log=1 OR
							ZTHL09.Status_Log=1 OR
							ZTHL10.Status_Log=1 OR
							ZTHL11.Status_Log=1 OR
							ZTHL12.Status_Log=1 OR
							ZTHL13.Status_Log=1 OR
							MODB01.Status_Log=1 OR
							MODB02.Status_Log=1 OR
							MBUS01.Status_Log=1,
							AllarmeLampada=>LAMP_AL
							);





			(* Test toggle *)
			(*IF TEST1 THEN TEST1:=FALSE; ELSE TEST1:=TRUE; END_IF*)
		END_IF

		Timer3(IN:=NOT Timer3.Q,PT:=T#5m);
		IF Timer3.Q THEN
			(* Trig logger *)
			LogTrig();
			(* Execute temporary CSV logger *)
			(*CSV_Log();*)
		END_IF

	S_SHUTDOWN:
		(* Stop sistema *)
		Sys.Status:=S_STARTUP;

	S_HALT:
		(* Aspetta uscita manuale *)
		Sys.Status:=S_STARTUP;

ELSE
	Sys.Status:=S_STARTUP;
END_CASE;
END_ACTION

(* POU Utils Functions/FLT_TAP, ST *)
FUNCTION_BLOCK FLT_TAP
VAR_INPUT
	IN		: BOOL;
	TAP		: BYTE:=4;
	INITEV	: BOOL:=TRUE;
END_VAR
VAR_OUTPUT
	OUT		: BOOL;
	EVH		: BOOL;
	EVL		: BOOL;
END_VAR
VAR
	init	: BOOL:=FALSE;
	cnt		: BYTE;
END_VAR
EVH:=FALSE;
EVL:=FALSE;

IF NOT init THEN
	init := TRUE;
	IF INITEV THEN
		OUT  := NOT IN;
		cnt  := TAP;
	ELSE
		OUT  := IN;
	END_IF
END_IF

IF OUT<>IN THEN
	cnt:=cnt+1;
	IF cnt>TAP THEN
		OUT:=IN;
		cnt:=0;
		IF OUT THEN EVH:=TRUE; ELSE EVL:=TRUE; END_IF
	END_IF
ELSE
	cnt:=0;
END_IF
END_FUNCTION_BLOCK

(* POU LON/Module_1/Module_1_PRG, FBD *)
PROGRAM Module_1_PRG
VAR
	(* Automatic added code, do not change! *)
	LonMaster : Module_1_LonMaster;
	SFPTnodeObject : Module_1_SFPTnodeObject;
	Virtualfunctionalblock : Module_1_Virtualfunctionalblock;

	InData_LON AT %IB0 : ARRAY[0..23] OF BYTE;
	OutData_LON AT %QB0 : ARRAY[0..23] OF BYTE;
	(***** End of automatic added code. *****)

	(* Add your code here. *)
	LonState: BOOL;
	LonReset: BOOL;

END_VAR
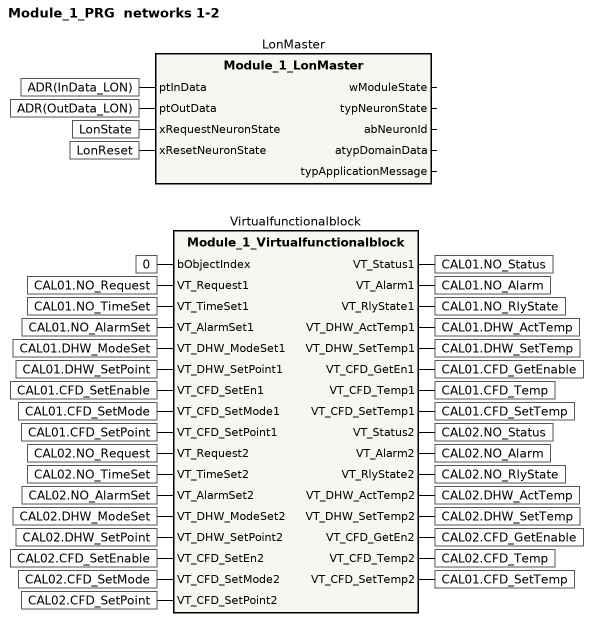
_FBD_ (* Function Block Diagram *)
NETWORK 1 (* Added by code generator *)
	LonMaster:Module_1_LonMaster(ptInData: ADR(InData_LON), ptOutData: ADR(OutData_LON), xRequestNeuronState: LonState, xResetNeuronState: LonReset)
NETWORK 2
	Virtualfunctionalblock:Module_1_Virtualfunctionalblock(bObjectIndex: 0, VT_Request1: CAL01.NO_Request, VT_TimeSet1: CAL01.NO_TimeSet, VT_AlarmSet1: CAL01.NO_AlarmSet, VT_DHW_ModeSet1: CAL01.DHW_ModeSet, VT_DHW_SetPoint1: CAL01.DHW_SetPoint, VT_CFD_SetEn1: CAL01.CFD_SetEnable, VT_CFD_SetMode1: CAL01.CFD_SetMode, VT_CFD_SetPoint1: CAL01.CFD_SetPoint, VT_Request2: CAL02.NO_Request, VT_TimeSet2: CAL02.NO_TimeSet, VT_AlarmSet2: CAL02.NO_AlarmSet, VT_DHW_ModeSet2: CAL02.DHW_ModeSet, VT_DHW_SetPoint2: CAL02.DHW_SetPoint, VT_CFD_SetEn2: CAL02.CFD_SetEnable, VT_CFD_SetMode2: CAL02.CFD_SetMode, VT_CFD_SetPoint2: CAL02.CFD_SetPoint, VT_Alarm1 => CAL01.NO_Alarm, VT_RlyState1 => CAL01.NO_RlyState, VT_DHW_ActTemp1 => CAL01.DHW_ActTemp, VT_DHW_SetTemp1 => CAL01.DHW_SetTemp, VT_CFD_GetEn1 => CAL01.CFD_GetEnable, VT_CFD_Temp1 => CAL01.CFD_Temp, VT_CFD_SetTemp1 => CAL01.CFD_SetTemp, VT_Status2 => CAL02.NO_Status, VT_Alarm2 => CAL02.NO_Alarm, VT_RlyState2 => CAL02.NO_RlyState, VT_DHW_ActTemp2 => CAL02.DHW_ActTemp, VT_DHW_SetTemp2 => CAL02.DHW_SetTemp, VT_CFD_GetEn2 => CAL02.CFD_GetEnable, VT_CFD_Temp2 => CAL02.CFD_Temp, VT_CFD_SetTemp2 => CAL01.CFD_SetTemp) => CAL01.NO_Status
_END_FBD_
(* the same logic as Structured Text *)
(* Network 1: Added by code generator *)
LonMaster(ptInData := ADR(InData_LON), ptOutData := ADR(OutData_LON), xRequestNeuronState := LonState, xResetNeuronState := LonReset);
(* Network 2 *)
Virtualfunctionalblock(bObjectIndex := 0, VT_Request1 := CAL01.NO_Request, VT_TimeSet1 := CAL01.NO_TimeSet, VT_AlarmSet1 := CAL01.NO_AlarmSet, VT_DHW_ModeSet1 := CAL01.DHW_ModeSet, VT_DHW_SetPoint1 := CAL01.DHW_SetPoint, VT_CFD_SetEn1 := CAL01.CFD_SetEnable, VT_CFD_SetMode1 := CAL01.CFD_SetMode, VT_CFD_SetPoint1 := CAL01.CFD_SetPoint, VT_Request2 := CAL02.NO_Request, VT_TimeSet2 := CAL02.NO_TimeSet, VT_AlarmSet2 := CAL02.NO_AlarmSet, VT_DHW_ModeSet2 := CAL02.DHW_ModeSet, VT_DHW_SetPoint2 := CAL02.DHW_SetPoint, VT_CFD_SetEn2 := CAL02.CFD_SetEnable, VT_CFD_SetMode2 := CAL02.CFD_SetMode, VT_CFD_SetPoint2 := CAL02.CFD_SetPoint);
CAL01.NO_Alarm := Virtualfunctionalblock.VT_Alarm1;
CAL01.NO_RlyState := Virtualfunctionalblock.VT_RlyState1;
CAL01.DHW_ActTemp := Virtualfunctionalblock.VT_DHW_ActTemp1;
CAL01.DHW_SetTemp := Virtualfunctionalblock.VT_DHW_SetTemp1;
CAL01.CFD_GetEnable := Virtualfunctionalblock.VT_CFD_GetEn1;
CAL01.CFD_Temp := Virtualfunctionalblock.VT_CFD_Temp1;
CAL01.CFD_SetTemp := Virtualfunctionalblock.VT_CFD_SetTemp1;
CAL02.NO_Status := Virtualfunctionalblock.VT_Status2;
CAL02.NO_Alarm := Virtualfunctionalblock.VT_Alarm2;
CAL02.NO_RlyState := Virtualfunctionalblock.VT_RlyState2;
CAL02.DHW_ActTemp := Virtualfunctionalblock.VT_DHW_ActTemp2;
CAL02.DHW_SetTemp := Virtualfunctionalblock.VT_DHW_SetTemp2;
CAL02.CFD_GetEnable := Virtualfunctionalblock.VT_CFD_GetEn2;
CAL02.CFD_Temp := Virtualfunctionalblock.VT_CFD_Temp2;
CAL01.CFD_SetTemp := Virtualfunctionalblock.VT_CFD_SetTemp2;
CAL01.NO_Status := Virtualfunctionalblock.VT_Status1;
END_PROGRAM

(* POU LON/Module_1/Master/Module_1_LonMaster, ST *)
FUNCTION_BLOCK Module_1_LonMaster
(******************************************)
(* Automatic generated code, do not edit! *)
(******************************************)
VAR_INPUT
	ptInData  : POINTER TO BYTE;
	ptOutData : POINTER TO BYTE;
	xRequestNeuronState : BOOL;
	xResetNeuronState : BOOL;
END_VAR
VAR_OUTPUT
	wModuleState : WORD; (* bit coded wModuleState:
	15: communication to I/O-module interrupted (error)
	14 - 08: reserved
	07: ready for Neuron initialization
	06: Neuron active
	05: user interface active
	04: internal module communication interrupted (error)
	03: CP synchronization running
	02: Neuron is configured online
	01 - 00: reserved *)

	typNeuronState : NeuronState;
	abNeuronId : ARRAY[0..5] OF BYTE;
	atypDomainData : ARRAY[0..1] OF DomainData;
	typApplicationMessage : ApplicationMessageData;
END_VAR
VAR
	bInternalCode : BYTE;
	bNvIndex : BYTE;
	wCpIndex : WORD;
	lonCom : FbLonBasicCommunication;

	xInitIsStarted : BOOL := FALSE;

	TimeoutTimer : TON;
	timeOutTime : TIME := T#1000ms;
	xStateMachineIsChecked : BOOL;
	xTimerStart : BOOL;

	iDomainTable : INT;
	xSendRequestPending : BOOL;
	trigRequest : R_TRIG;
	trigReset : R_TRIG;

	abMbxRxPrio0Buf: ARRAY [0..309] OF BYTE;
	abMbxRxPrio1Buf: ARRAY [0..517] OF BYTE;
	aMbxRxBufSize: ARRAY [0..1] OF UINT := 310, 518;
	aMbxRxBufList: ARRAY [0..1] OF POINTER TO BYTE;
	afbMbxRxFb: ARRAY [0..1] OF MBX2_RX_DEFRAG;
	astMbxRxCtx: ARRAY [0..1] OF stMbx2DefragContext;

	abMbxTxPrio0Buf: ARRAY [0..309] OF BYTE;
	abMbxTxPrio1Buf: ARRAY [0..517] OF BYTE;
	aMbxTxBufSize: ARRAY [0..1] OF UINT := 310, 518;
	aMbxTxBufList: ARRAY [0..1] OF POINTER TO BYTE;
	afbMbxTxFb: ARRAY [0..1] OF MBX2_TX_FRAG;

	astMbxTrackContext: ARRAY [0..0] OF stMbx2TrackContext;
END_VAR
VAR CONSTANT
END_VAR
aMbxRxBufList[0] := ADR(abMbxRxPrio0Buf[0]);
aMbxRxBufList[1] := ADR(abMbxRxPrio1Buf[0]);

aMbxTxBufList[0] := ADR(abMbxTxPrio0Buf[0]);
aMbxTxBufList[1] := ADR(abMbxTxPrio1Buf[0]);

mbxModule_1.Ressources.pDefragBufList := ADR(aMbxRxBufList);
mbxModule_1.Ressources.pDefragBufSizeList := ADR(aMbxRxBufSize);
mbxModule_1.Ressources.pDefragCtxPtrList := ADR(astMbxRxCtx);
mbxModule_1.Ressources.pDefragFbList := ADR(afbMbxRxFb);
mbxModule_1.Ressources.pFragBufList := ADR(aMbxTxBufList);
mbxModule_1.Ressources.pFragBufSizeList := ADR(aMbxTxBufSize);
mbxModule_1.Ressources.pFragFbList := ADR(afbMbxTxFb);

mbxModule_1.Ressources.unMaxAvailableRxPrioIndex := 1;
mbxModule_1.Ressources.unMaxAvailableTxPrioIndex := 1;

mbxModule_1.Ressources.pTrackStList := ADR(astMbxTrackContext);
mbxModule_1.Ressources.unMaxAvailableTrackIndex := 0;

mbxModule_1.Ressources.pabRxWin := ptInData + 1;
mbxModule_1.Ressources.pabTxWin := ptOutData + 1;
mbxModule_1.Ressources.bTxWinSize := 23;
mbxModule_1.Ressources.bRxWinSize := 23;

IF (mbxModule_1.bStatus.2 = TRUE) OR (mbxModule_1.bStatus.1 = TRUE) THEN
	mbxModule_1.MBX_RESET();
	xInitRunning_Module_1 := TRUE;
	xInitIsStarted := FALSE;
END_IF
mbxModule_1.MBX_CYCLE();

IF (mbxModule_1.bStatus.0 <> TRUE) THEN 
	wModuleState := 16#8000;
	RETURN;
ELSE
	wModuleState.15 := FALSE;
END_IF

xStateMachineIsChecked := FALSE;
IF xInitRunning_Module_1 = TRUE THEN
	IF xInitIsStarted = FALSE THEN
		SetParameter();
		lonCom.eInitState := INIT_SND_SGNTR_REQ;
		lonCom.CheckInitState();
		xInitIsStarted := TRUE;
		xStateMachineIsChecked := TRUE;
	END_IF
END_IF

typApplicationMessage.xMsgRcvd := FALSE;
typApplicationMessage.xRspRcvd := FALSE;
ResetNviUpdate();
WHILE (mbxModule_1.xRxPending) DO
	unLastLen_mbxModule_1 := mbxModule_1.unRxLen;
	mbxModule_1.pbRxData := ADR(InDataTelegram_Module_1);
	mbxModule_1.MBX_RETRIEVE();
	IF (mbxModule_1.nError <> MBX_OK) THEN EXIT; END_IF;
	bInternalCode := InDataTelegram_Module_1[0];

	IF (xInitRunning_Module_1 = TRUE) AND (lonCom.eInitState <> INIT_TRANSFER_CFG) THEN
		IF (FuCheckForValidInitCode(bInternalCode)) THEN
			SetParameter();
			lonCom.unLastLen := unLastLen_mbxModule_1;
			lonCom.CheckInitState();
			xInitRunning_Module_1 := NOT lonCom.xInitDone;
			xStateMachineIsChecked := TRUE;
		END_IF
	END_IF

	IF (bInternalCode = M2C_NVI_UPDT_OCCD) OR (bInternalCode = M2C_NV_VALUE_RSP) OR (bInternalCode = M2C_NVI_UPDT_TOUT) THEN
		bNvIndex := InDataTelegram_Module_1[1];
		CASE bNvIndex OF
			0, 2, 4: Module_1_PRG.SFPTnodeObject.DataReceived();
			6, 8, 10, 12, 14, 16, 18, 20, 22, 24, 26, 28, 30, 32, 34, 36: Module_1_PRG.Virtualfunctionalblock.DataReceived();

		END_CASE;
	ELSIF (bInternalCode = M2C_CP_VALUE_RSP) THEN
		wCpIndex := InDataTelegram_Module_1[1] OR (InDataTelegram_Module_1[2] * 256);
		CASE wCpIndex OF

		END_CASE;
	ELSIF (bInternalCode = M2C_LON_MSG_RCVD) OR (bInternalCode = M2C_LON_RSP_RCVD) THEN
		ApplMsgReceived();
	ELSIF (bInternalCode = M2C_STATUS_RSP) THEN
		wModuleState := (wModuleState AND 16#FF00) + InDataTelegram_Module_1[1];
	ELSIF (bInternalCode = M2C_NEURON_ID) THEN
		FuMemCopy(ADR(InDataTelegram_Module_1[1]), ADR(abNeuronId), 6);
	ELSIF (bInternalCode = M2C_DOMAIN_DATA) THEN
		DomainDataRcvd();
	ELSIF (bInternalCode = M2C_MICRO_SERVER_STATUS_RSP) THEN
		NeuronStateRcvd();
	END_IF
END_WHILE

IF (xInitRunning_Module_1 = TRUE) AND ((lonCom.xCallStateMachine = TRUE) OR (TimeoutTimer.Q = TRUE)) AND (NOT xStateMachineIsChecked) THEN
	SetParameter();
	lonCom.xTimeOut := TimeoutTimer.Q;
	lonCom.CheckInitState();
END_IF
TimeoutTimer(IN:=lonCom.xTimerStart, PT:=timeOutTime);

trigRequest(CLK := xRequestNeuronState);
trigReset(CLK := xResetNeuronState);
IF (trigRequest.Q OR trigReset.Q) THEN
	RequestNeuronState();
END_IF
END_FUNCTION_BLOCK
ACTION ApplMsgReceived:
IF (InDataTelegram_Module_1[0] = M2C_LON_MSG_RCVD) THEN
	typApplicationMessage.typService := InDataTelegram_Module_1[1] AND 16#30;
	typApplicationMessage.bSourceSubnetId := InDataTelegram_Module_1[2];
	typApplicationMessage.bSourceNodeId := InDataTelegram_Module_1[3];
	typApplicationMessage.bCorrelator := InDataTelegram_Module_1[4];
	typApplicationMessage.bCode :=  InDataTelegram_Module_1[5];
	typApplicationMessage.bDataLength := UINT_TO_BYTE(unLastLen_mbxModule_1 - 6);
	IF typApplicationMessage.bDataLength > 48 THEN typApplicationMessage.bDataLength := 48; END_IF;
	FuMemSet(ADR(typApplicationMessage.abData), 0, SIZEOF(typApplicationMessage.abData));
	IF typApplicationMessage.bDataLength > 0 THEN
		FuMemCopy(ADR(InDataTelegram_Module_1[6]), ADR(typApplicationMessage.abData), typApplicationMessage.bDataLength);
	END_IF
	typApplicationMessage.xMsgRcvd := TRUE;
ELSE
	typApplicationMessage.typService := LON_RESPONSE;
	typApplicationMessage.bSourceSubnetId := InDataTelegram_Module_1[1];
	typApplicationMessage.bSourceNodeId := InDataTelegram_Module_1[2];
	typApplicationMessage.bCorrelator := 0;
	typApplicationMessage.bCode :=  InDataTelegram_Module_1[3];
	typApplicationMessage.bDataLength := UINT_TO_BYTE(unLastLen_mbxModule_1 - 4);
	IF typApplicationMessage.bDataLength > 48 THEN typApplicationMessage.bDataLength := 48; END_IF;
	FuMemSet(ADR(typApplicationMessage.abData), 0, SIZEOF(typApplicationMessage.abData));
	IF typApplicationMessage.bDataLength > 0 THEN
		FuMemCopy(ADR(InDataTelegram_Module_1[4]), ADR(typApplicationMessage.abData), typApplicationMessage.bDataLength);
	END_IF
	typApplicationMessage.xRspRcvd := TRUE;
END_IF
END_ACTION
ACTION DomainDataRcvd:
IF (unLastLen_mbxModule_1 = 17) THEN
	iDomainTable := InDataTelegram_Module_1[1];
	IF (iDomainTable < 0) OR (iDomainTable > 1) THEN RETURN; END_IF
	FuMemCopy(ADR(InDataTelegram_Module_1[2]), ADR(atypDomainData[iDomainTable].abDomainId), 6);
	atypDomainData[iDomainTable].bSubnet := InDataTelegram_Module_1[8];
	atypDomainData[iDomainTable].xIsNonClone := InDataTelegram_Module_1[9].7;
	atypDomainData[iDomainTable].bNodeId := InDataTelegram_Module_1[9] AND 16#7F;
	atypDomainData[iDomainTable].xIsInvalid := InDataTelegram_Module_1[10].7;
	atypDomainData[iDomainTable].bDomainIdLength := InDataTelegram_Module_1[10] AND 16#7F;
	FuMemCopy(ADR(InDataTelegram_Module_1[11]), ADR(atypDomainData[iDomainTable].abAuthenticationKey), 6);
END_IF
END_ACTION
ACTION NeuronStateRcvd:
IF (unLastLen_mbxModule_1 = 16) THEN
	typNeuronState.wCrcError := InDataTelegram_Module_1[1] + InDataTelegram_Module_1[2] * 256;
	typNeuronState.wTransactionTimeouts := InDataTelegram_Module_1[3] + InDataTelegram_Module_1[4] * 256;
	typNeuronState.wReceiveTransactionBuffersFull := InDataTelegram_Module_1[5] + InDataTelegram_Module_1[6] * 256;
	typNeuronState.wLostMessages := InDataTelegram_Module_1[7] + InDataTelegram_Module_1[8] * 256;
	typNeuronState.wMissedMessages := InDataTelegram_Module_1[9] + InDataTelegram_Module_1[10] * 256;
	typNeuronState.bResetCause := InDataTelegram_Module_1[11];
	typNeuronState.bNodeState := InDataTelegram_Module_1[12];
	typNeuronState.bFirmwareVersion := InDataTelegram_Module_1[13];
	typNeuronState.bLastErrorLogged := InDataTelegram_Module_1[14];
	typNeuronState.bModelNumber := InDataTelegram_Module_1[15];
END_IF
END_ACTION
ACTION RequestNeuronState:
OutDataTelegram_Module_1[0] := C2M_MICRO_SERVER_STATUS_QRY;
OutDataTelegram_Module_1[1] := BOOL_TO_BYTE(trigReset.Q);

mbxModule_1.bTxPrio := 1;
mbxModule_1.bTxProtID := 0;
mbxModule_1.pbTxData := ADR(OutDataTelegram_Module_1);
mbxModule_1.unTxLen := 2;
mbxModule_1.MBX_SEND();

IF (mbxModule_1.nError <> MBX_OK) THEN
	RETURN;
END_IF
END_ACTION
ACTION ResetNviUpdate:
Module_1_PRG.SFPTnodeObject.ResetNviUpdate();
Module_1_PRG.Virtualfunctionalblock.ResetNviUpdate();
END_ACTION
ACTION SetParameter:
lonCom.pMbx 			:= ADR(mbxModule_1);
lonCom.pInData 			:= ADR(InDataTelegram_Module_1);
lonCom.pOutData 		:= ADR(OutDataTelegram_Module_1);
lonCom.pTimer			:= ADR(TimeoutTimer);

lonCom.pActualSignature	:= ADR(abSignature_Module_1);
lonCom.pConfigBlock := ADR(abInterface_Module_1);
lonCom.wConfigSize 		:= wConfigSize_Module_1;
END_ACTION

(* POU LON/Module_1/NV_Interface/Module_1_SFPTnodeObject, ST *)
FUNCTION_BLOCK Module_1_SFPTnodeObject
(******************************************)
(* Automatic generated code, do not edit! *)
(******************************************)
VAR_INPUT
	bObjectIndex : BYTE := 0;
	nvoStatus : typSnvtObjStatus;
	nvoFileStat : typSnvtFileStatus;

END_VAR
VAR_OUTPUT
	nviRequest : typSnvtObjRequest;
	nviFileReq : typSnvtFileReq;
	nviFilePos : typSnvtFilePos;

END_VAR
VAR
	xSetOnce : BOOL := TRUE;
	xDataInUpdated : BOOL := FALSE;
	nvoStatusLast: typSnvtObjStatus;
	nvoFileStatLast: typSnvtFileStatus;

	cmd : BYTE;
	z : INT;
	bNvRelativeIdx : BYTE;
	bNvAbsoluteIdx : BYTE;
	wCpRelativeIdx : WORD;
	wCpAbsoluteIdx : WORD;
END_VAR
VAR CONSTANT
	bNvStartIndex : BYTE := 0;
	wCpStartIndex : WORD := 65535;
	bLmoCount : BYTE := 1;
END_VAR
IF (xInitRunning_Module_1 = TRUE) AND (xSetOnce = TRUE) THEN
	xSetOnce := FALSE;
	CachePointers();
	SetUpdateFlags();
END_IF

CheckUpdateFlags();
IF (xInitRunning_Module_1 = FALSE) AND (xDataInUpdated = FALSE) THEN
	IF (mbxModule_1.bStatus.0) THEN
		SendValueRequest();
	END_IF
END_IF

IF (xInitRunning_Module_1 = FALSE) AND (mbxModule_1.bStatus.0) THEN
	xSetOnce := TRUE;
	xDataInUpdated := FALSE;
	IF ((NOT FuMemCompare(ADR(nvoStatusLast), ADR(nvoStatus), ADR(nvoStatus.bStatusInformation) - ADR(nvoStatus))) OR (nvoStatus.bStatusInformation.7 = TRUE) OR (nvoStatusLast.bInternalUseOnly.1 = TRUE)) THEN
		FuSnvtObjStatusToRaw(ADR(nvoStatus), ADR(OutDataTelegram_Module_1[2]));

		bNvAbsoluteIdx := bNvStartIndex + bObjectIndex + (1 * bLmoCount);

		IF (FuDoNvoUpdate_Module_1(ADR(nvoStatus), ADR(nvoStatusLast), ADR(nvoStatus.bInternalUseOnly), ADR(nvoStatusLast.bInternalUseOnly), ADR(nvoStatus.bStatusInformation), bNvAbsoluteIdx, 6, SIZEOF(nvoStatus)) = FALSE) THEN
			RETURN;
		END_IF
	END_IF
	IF ((NOT FuMemCompare(ADR(nvoFileStatLast), ADR(nvoFileStat), ADR(nvoFileStat.bStatusInformation) - ADR(nvoFileStat))) OR (nvoFileStat.bStatusInformation.7 = TRUE) OR (nvoFileStatLast.bInternalUseOnly.1 = TRUE)) THEN
		FuSnvtFileStatusToRaw(ADR(nvoFileStat), ADR(OutDataTelegram_Module_1[2]));

		bNvAbsoluteIdx := bNvStartIndex + bObjectIndex + (3 * bLmoCount);

		IF (FuDoNvoUpdate_Module_1(ADR(nvoFileStat), ADR(nvoFileStatLast), ADR(nvoFileStat.bInternalUseOnly), ADR(nvoFileStatLast.bInternalUseOnly), ADR(nvoFileStat.bStatusInformation), bNvAbsoluteIdx, 27, SIZEOF(nvoFileStat)) = FALSE) THEN
			RETURN;
		END_IF
	END_IF

END_IF
END_FUNCTION_BLOCK
ACTION CachePointers:
;
END_ACTION
ACTION CheckUpdateFlags:
xDataInUpdated := (NOT nviRequest.bInternalUseOnly.0) AND (NOT nviFileReq.bInternalUseOnly.0) AND (NOT nviFilePos.bInternalUseOnly.0) AND TRUE;
END_ACTION
ACTION DataReceived:
cmd := InDataTelegram_Module_1[0];
IF (cmd = M2C_NVI_UPDT_OCCD) OR (cmd = M2C_NV_VALUE_RSP) OR (cmd = M2C_NVI_UPDT_TOUT) THEN
	bNvRelativeIdx := (InDataTelegram_Module_1[1] - bNvStartIndex - bObjectIndex) / bLmoCount;
	CASE bNvRelativeIdx OF
	0:
		IF (cmd = M2C_NVI_UPDT_OCCD) OR (cmd = M2C_NV_VALUE_RSP) THEN
			IF (unLastLen_mbxModule_1 = (2 + 3)) THEN
				FuRawToSnvtObjRequest(ADR(InDataTelegram_Module_1[2]), ADR(nviRequest));
				nviRequest.bInternalUseOnly.0 := FALSE;
				nviRequest.bStatusInformation := FuInkrementNviStatus(nviRequest.bStatusInformation);
			ELSIF (unLastLen_mbxModule_1 = 2) THEN
				nviRequest.bStatusInformation := FuInkrementNviStatus(nviRequest.bStatusInformation);
			END_IF
		ELSIF (cmd = M2C_NVI_UPDT_TOUT) THEN
			IF (unLastLen_mbxModule_1 = 3) THEN
				nviRequest.bStatusInformation.4 := BYTE_TO_BOOL(InDataTelegram_Module_1[2]);
			END_IF
		END_IF
	2:
		IF (cmd = M2C_NVI_UPDT_OCCD) OR (cmd = M2C_NV_VALUE_RSP) THEN
			IF (unLastLen_mbxModule_1 = (2 + 12)) THEN
				FuRawToSnvtFileReq(ADR(InDataTelegram_Module_1[2]), ADR(nviFileReq));
				nviFileReq.bInternalUseOnly.0 := FALSE;
				nviFileReq.bStatusInformation := FuInkrementNviStatus(nviFileReq.bStatusInformation);
			ELSIF (unLastLen_mbxModule_1 = 2) THEN
				nviFileReq.bStatusInformation := FuInkrementNviStatus(nviFileReq.bStatusInformation);
			END_IF
		ELSIF (cmd = M2C_NVI_UPDT_TOUT) THEN
			IF (unLastLen_mbxModule_1 = 3) THEN
				nviFileReq.bStatusInformation.4 := BYTE_TO_BOOL(InDataTelegram_Module_1[2]);
			END_IF
		END_IF
	4:
		IF (cmd = M2C_NVI_UPDT_OCCD) OR (cmd = M2C_NV_VALUE_RSP) THEN
			IF (unLastLen_mbxModule_1 = (2 + 6)) THEN
				FuRawToSnvtFilePos(ADR(InDataTelegram_Module_1[2]), ADR(nviFilePos));
				nviFilePos.bInternalUseOnly.0 := FALSE;
				nviFilePos.bStatusInformation := FuInkrementNviStatus(nviFilePos.bStatusInformation);
			ELSIF (unLastLen_mbxModule_1 = 2) THEN
				nviFilePos.bStatusInformation := FuInkrementNviStatus(nviFilePos.bStatusInformation);
			END_IF
		ELSIF (cmd = M2C_NVI_UPDT_TOUT) THEN
			IF (unLastLen_mbxModule_1 = 3) THEN
				nviFilePos.bStatusInformation.4 := BYTE_TO_BOOL(InDataTelegram_Module_1[2]);
			END_IF
		END_IF

	END_CASE
ELSIF (cmd = M2C_CP_VALUE_RSP) THEN
	wCpRelativeIdx := ((InDataTelegram_Module_1[1] + InDataTelegram_Module_1[2] * 256) - wCpStartIndex - bObjectIndex) / bLmoCount;
	CASE wCpRelativeIdx OF

	END_CASE
END_IF
END_ACTION
ACTION ResetNviUpdate:
nviRequest.bStatusInformation := nviRequest.bStatusInformation AND 16#F8;
nviFileReq.bStatusInformation := nviFileReq.bStatusInformation AND 16#F8;
nviFilePos.bStatusInformation := nviFilePos.bStatusInformation AND 16#F8;
;
END_ACTION
ACTION SendValueRequest:
IF (FuSendNviValueReq_Module_1(ADR(nviRequest.bInternalUseOnly), bNvStartIndex + bObjectIndex + (0 * bLmoCount)) = FALSE) THEN
	RETURN;
END_IF

IF (FuSendNviValueReq_Module_1(ADR(nviFileReq.bInternalUseOnly), bNvStartIndex + bObjectIndex + (2 * bLmoCount)) = FALSE) THEN
	RETURN;
END_IF

IF (FuSendNviValueReq_Module_1(ADR(nviFilePos.bInternalUseOnly), bNvStartIndex + bObjectIndex + (4 * bLmoCount)) = FALSE) THEN
	RETURN;
END_IF

;
END_ACTION
ACTION SetUpdateFlags:
nviRequest.bInternaluseOnly.0 := TRUE;
nvoStatusLast.bInternaluseOnly.1 := TRUE;
nvoStatusLast.bInternaluseOnly.7 := FALSE;
nviFileReq.bInternaluseOnly.0 := TRUE;
nvoFileStatLast.bInternaluseOnly.1 := TRUE;
nvoFileStatLast.bInternaluseOnly.7 := FALSE;
nviFilePos.bInternaluseOnly.0 := TRUE;
;
END_ACTION

(* POU LON/Shared/Internal/FuSnvtObjStatusToRaw, ST *)
FUNCTION FuSnvtObjStatusToRaw : BOOL
(******************************************)
(* Automatic generated code, do not edit! *)
(******************************************)
VAR_INPUT
	NvDataIn :  POINTER TO typSnvtObjStatus;
	DataOut : POINTER TO ARRAY[0..5] OF BYTE;
END_VAR
VAR
END_VAR
DataOut^[0] := WORD_TO_BYTE(SHR(NvDataIn^.wObjectId, 8));
DataOut^[1] := WORD_TO_BYTE(NvDataIn^.wObjectId);

DataOut^[2] := NvDataIn^.bBitfieldByteOffset2;

DataOut^[3] := NvDataIn^.bBitfieldByteOffset3;

DataOut^[4] := NvDataIn^.bBitfieldByteOffset4;

DataOut^[5] := NvDataIn^.bBitfieldByteOffset5;

FuSnvtObjStatusToRaw := TRUE;
END_FUNCTION

(* POU LON/Module_1/Internal/FuDoNvoUpdate_Module_1, ST *)
FUNCTION FuDoNvoUpdate_Module_1 : BOOL
(******************************************)
(* Automatic generated code, do not edit! *)
(******************************************)
VAR_INPUT
	ptNvo : POINTER TO BYTE;
	ptNvoLast : POINTER TO BYTE;
	ptNvoInternalUse : POINTER TO BYTE;
	ptNvoLastInternalUse : POINTER TO BYTE;
	ptNvoStatusInformation : POINTER TO BYTE;
	bNvoIndex : BYTE;
	uiNvoLength : UINT;
	uiNvoVariableLength : UINT;
END_VAR
IF (ptNvoLastInternalUse^.1 = TRUE) AND (ptNvoStatusInformation^.7 = FALSE) THEN
	OutDataTelegram_Module_1[0] := C2M_NV_VALUE;
ELSE
	OutDataTelegram_Module_1[0] := C2M_NVO_PROPAGATE;
END_IF
OutDataTelegram_Module_1[1] := bNvoIndex;

mbxModule_1.bTxPrio := BOOL_TO_BYTE(ptNvoLastInternalUse^.7);
mbxModule_1.bTxProtID := 0;
mbxModule_1.pbTxData := ADR(OutDataTelegram_Module_1);
mbxModule_1.unTxLen := 2 + uiNvoLength;
mbxModule_1.MBX_SEND();

IF (mbxModule_1.nError <> MBX_OK) THEN
	FuDoNvoUpdate_Module_1 := FALSE;
	RETURN;
END_IF

ptNvoLastInternalUse^.1 := FALSE;
ptNvoInternalUse^ := ptNvoLastInternalUse^;
FuMemCopy(ptNvo, ptNvoLast, uiNvoVariableLength);

FuDoNvoUpdate_Module_1 := TRUE;
END_FUNCTION

(* POU LON/Shared/Internal/FuSnvtFileStatusToRaw, ST *)
FUNCTION FuSnvtFileStatusToRaw : BOOL
(******************************************)
(* Automatic generated code, do not edit! *)
(******************************************)
VAR_INPUT
	NvDataIn :  POINTER TO typSnvtFileStatus;
	DataOut : POINTER TO ARRAY[0..26] OF BYTE;
END_VAR
VAR
END_VAR
DataOut^[0] := NvDataIn^.bStatus;

DataOut^[1] := WORD_TO_BYTE(SHR(NvDataIn^.wNumberOfFiles, 8));
DataOut^[2] := WORD_TO_BYTE(NvDataIn^.wNumberOfFiles);

DataOut^[3] := WORD_TO_BYTE(SHR(NvDataIn^.wSelectedFile, 8));
DataOut^[4] := WORD_TO_BYTE(NvDataIn^.wSelectedFile);

DataOut^[5] := NvDataIn^.abAdr[0];
DataOut^[6] := NvDataIn^.abAdr[1];
DataOut^[7] := NvDataIn^.abAdr[2];
DataOut^[8] := NvDataIn^.abAdr[3];
DataOut^[9] := NvDataIn^.abAdr[4];
DataOut^[10] := NvDataIn^.abAdr[5];
DataOut^[11] := NvDataIn^.abAdr[6];
DataOut^[12] := NvDataIn^.abAdr[7];
DataOut^[13] := NvDataIn^.abAdr[8];
DataOut^[14] := NvDataIn^.abAdr[9];
DataOut^[15] := NvDataIn^.abAdr[10];
DataOut^[16] := NvDataIn^.abAdr[11];
DataOut^[17] := NvDataIn^.abAdr[12];
DataOut^[18] := NvDataIn^.abAdr[13];
DataOut^[19] := NvDataIn^.abAdr[14];
DataOut^[20] := NvDataIn^.abAdr[15];
DataOut^[21] := NvDataIn^.abAdr[16];
DataOut^[22] := NvDataIn^.abAdr[17];
DataOut^[23] := NvDataIn^.abAdr[18];
DataOut^[24] := NvDataIn^.abAdr[19];
DataOut^[25] := NvDataIn^.abAdr[20];
DataOut^[26] := NvDataIn^.abAdr[21];

FuSnvtFileStatusToRaw := TRUE;
END_FUNCTION

(* POU LON/Module_1/Internal/FuSendNviValueReq_Module_1, ST *)
FUNCTION FuSendNviValueReq_Module_1 : BOOL
(******************************************)
(* Automatic generated code, do not edit! *)
(******************************************)
VAR_INPUT
	ptInternalUseOnly : POINTER TO BYTE;
	bNvIndex : BYTE;
END_VAR
IF ptInternalUseOnly^.0 = TRUE THEN
	OutDataTelegram_Module_1[0] := C2M_NV_VALUE_QRY;
	OutDataTelegram_Module_1[1] := bNvIndex;

	mbxModule_1.bTxPrio := 1;
	mbxModule_1.bTxProtID := 0;
	mbxModule_1.pbTxData := ADR(OutDataTelegram_Module_1);
	mbxModule_1.unTxLen := 2;
	mbxModule_1.MBX_SEND();

	IF (mbxModule_1.nError <> MBX_OK) THEN
		FuSendNviValueReq_Module_1 := FALSE;
		RETURN;
	END_IF
	ptInternalUseOnly^.0 := FALSE;
END_IF

FuSendNviValueReq_Module_1 := TRUE;
END_FUNCTION

(* POU LON/Module_1/NV_Interface/Module_1_Virtualfunctionalblock, ST *)
FUNCTION_BLOCK Module_1_Virtualfunctionalblock
(******************************************)
(* Automatic generated code, do not edit! *)
(******************************************)
VAR_INPUT
	bObjectIndex : BYTE := 0;
	VT_Request1 : typSnvtObjRequest;
	VT_TimeSet1 : typSnvtTimeStamp;
	VT_AlarmSet1 : typSnvtAlarm;
	VT_DHW_ModeSet1 : typSnvtHvacMode;
	VT_DHW_SetPoint1 : typSnvtTempP;
	VT_CFD_SetEn1 : typSnvtSwitch;
	VT_CFD_SetMode1 : typSnvtHvacMode;
	VT_CFD_SetPoint1 : typSnvtTempP;
	VT_Request2 : typSnvtObjRequest;
	VT_TimeSet2 : typSnvtTimeStamp;
	VT_AlarmSet2 : typSnvtAlarm;
	VT_DHW_ModeSet2 : typSnvtHvacMode;
	VT_DHW_SetPoint2 : typSnvtTempP;
	VT_CFD_SetEn2 : typSnvtSwitch;
	VT_CFD_SetMode2 : typSnvtHvacMode;
	VT_CFD_SetPoint2 : typSnvtTempP;

END_VAR
VAR_OUTPUT
	VT_Status1 : typSnvtObjStatus;
	VT_Alarm1 : typSnvtAlarm;
	VT_RlyState1 : typSnvtState;
	VT_DHW_ActTemp1 : typSnvtTempP;
	VT_DHW_SetTemp1 : typSnvtTempP;
	VT_CFD_GetEn1 : typSnvtSwitch;
	VT_CFD_Temp1 : typSnvtTempP;
	VT_CFD_SetTemp1 : typSnvtTempP;
	VT_Status2 : typSnvtObjStatus;
	VT_Alarm2 : typSnvtAlarm;
	VT_RlyState2 : typSnvtState;
	VT_DHW_ActTemp2 : typSnvtTempP;
	VT_DHW_SetTemp2 : typSnvtTempP;
	VT_CFD_GetEn2 : typSnvtSwitch;
	VT_CFD_Temp2 : typSnvtTempP;
	VT_CFD_SetTemp2 : typSnvtTempP;

END_VAR
VAR
	xSetOnce : BOOL := TRUE;
	xDataInUpdated : BOOL := FALSE;
	paNviSnvtObjStatus : ARRAY[0..1] OF POINTER TO typSnvtObjStatus;
	aNviSnvtObjStatusIndex : ARRAY[0..1] OF BYTE := 1,17;
	paNviSnvtAlarm : ARRAY[0..1] OF POINTER TO typSnvtAlarm;
	aNviSnvtAlarmIndex : ARRAY[0..1] OF BYTE := 3,19;
	paNviSnvtState : ARRAY[0..1] OF POINTER TO typSnvtState;
	aNviSnvtStateIndex : ARRAY[0..1] OF BYTE := 5,21;
	paNviSnvtTempP : ARRAY[0..7] OF POINTER TO typSnvtTempP;
	aNviSnvtTempPIndex : ARRAY[0..7] OF BYTE := 7,9,13,15,23,25,29,31;
	paNviSnvtSwitch : ARRAY[0..1] OF POINTER TO typSnvtSwitch;
	aNviSnvtSwitchIndex : ARRAY[0..1] OF BYTE := 11,27;
	paNvoSnvtObjRequest : ARRAY[0..1] OF POINTER TO typSnvtObjRequest;
	aNvoSnvtObjRequestIndex : ARRAY[0..1] OF BYTE := 0,16;
	aNvoSnvtObjRequestLast : ARRAY[0..1] OF typSnvtObjRequest;
	aNvoSnvtObjRequestPriority : ARRAY[0..0] OF BYTE := 16#00;
	paNvoSnvtTimeStamp : ARRAY[0..1] OF POINTER TO typSnvtTimeStamp;
	aNvoSnvtTimeStampIndex : ARRAY[0..1] OF BYTE := 2,18;
	aNvoSnvtTimeStampLast : ARRAY[0..1] OF typSnvtTimeStamp;
	aNvoSnvtTimeStampPriority : ARRAY[0..0] OF BYTE := 16#00;
	paNvoSnvtAlarm : ARRAY[0..1] OF POINTER TO typSnvtAlarm;
	aNvoSnvtAlarmIndex : ARRAY[0..1] OF BYTE := 4,20;
	aNvoSnvtAlarmLast : ARRAY[0..1] OF typSnvtAlarm;
	aNvoSnvtAlarmPriority : ARRAY[0..0] OF BYTE := 16#00;
	paNvoSnvtHvacMode : ARRAY[0..3] OF POINTER TO typSnvtHvacMode;
	aNvoSnvtHvacModeIndex : ARRAY[0..3] OF BYTE := 6,12,22,28;
	aNvoSnvtHvacModeLast : ARRAY[0..3] OF typSnvtHvacMode;
	aNvoSnvtHvacModePriority : ARRAY[0..0] OF BYTE := 16#00;
	paNvoSnvtTempP : ARRAY[0..3] OF POINTER TO typSnvtTempP;
	aNvoSnvtTempPIndex : ARRAY[0..3] OF BYTE := 8,14,24,30;
	aNvoSnvtTempPLast : ARRAY[0..3] OF typSnvtTempP;
	aNvoSnvtTempPPriority : ARRAY[0..0] OF BYTE := 16#00;
	paNvoSnvtSwitch : ARRAY[0..1] OF POINTER TO typSnvtSwitch;
	aNvoSnvtSwitchIndex : ARRAY[0..1] OF BYTE := 10,26;
	aNvoSnvtSwitchLast : ARRAY[0..1] OF typSnvtSwitch;
	aNvoSnvtSwitchPriority : ARRAY[0..0] OF BYTE := 16#00;

	cmd : BYTE;
	z : INT;
	bNvRelativeIdx : BYTE;
	bNvAbsoluteIdx : BYTE;
	wCpRelativeIdx : WORD;
	wCpAbsoluteIdx : WORD;
END_VAR
VAR CONSTANT
	bNvStartIndex : BYTE := 5;
	wCpStartIndex : WORD := 65535;
	bLmoCount : BYTE := 1;
END_VAR
IF (xInitRunning_Module_1 = TRUE) AND (xSetOnce = TRUE) THEN
	xSetOnce := FALSE;
	CachePointers();
	SetUpdateFlags();
END_IF

CheckUpdateFlags();
IF (xInitRunning_Module_1 = FALSE) AND (xDataInUpdated = FALSE) THEN
	IF (mbxModule_1.bStatus.0) THEN
		SendValueRequest();
	END_IF
END_IF

IF (xInitRunning_Module_1 = FALSE) AND (mbxModule_1.bStatus.0) THEN
	xSetOnce := TRUE;
	xDataInUpdated := FALSE;
	FOR z := 0 TO 1 DO
		IF ((NOT FuMemCompare(ADR(aNvoSnvtObjRequestLast[z]), paNvoSnvtObjRequest[z], ADR(paNvoSnvtObjRequest[z]^.bStatusInformation) - paNvoSnvtObjRequest[z])) OR (paNvoSnvtObjRequest[z]^.bStatusInformation.7 = TRUE) OR (aNvoSnvtObjRequestLast[z].bInternalUseOnly.1 = TRUE)) THEN
			FuSnvtObjRequestToRaw(paNvoSnvtObjRequest[z], ADR(OutDataTelegram_Module_1[2]));

			bNvAbsoluteIdx := bNvStartIndex + bObjectIndex + (aNvoSnvtObjRequestIndex[z] * bLmoCount);

			IF (FuDoNvoUpdate_Module_1(paNvoSnvtObjRequest[z], ADR(aNvoSnvtObjRequestLast[z]), ADR(paNvoSnvtObjRequest[z]^.bInternalUseOnly), ADR(aNvoSnvtObjRequestLast[z].bInternalUseOnly), ADR(paNvoSnvtObjRequest[z]^.bStatusInformation), bNvAbsoluteIdx, 3, SIZEOF(aNvoSnvtObjRequestLast[z])) = FALSE) THEN
				RETURN;
			END_IF
		END_IF
	END_FOR
	FOR z := 0 TO 1 DO
		IF ((NOT FuMemCompare(ADR(aNvoSnvtTimeStampLast[z]), paNvoSnvtTimeStamp[z], ADR(paNvoSnvtTimeStamp[z]^.bStatusInformation) - paNvoSnvtTimeStamp[z])) OR (paNvoSnvtTimeStamp[z]^.bStatusInformation.7 = TRUE) OR (aNvoSnvtTimeStampLast[z].bInternalUseOnly.1 = TRUE)) THEN
			FuSnvtTimeStampToRaw(paNvoSnvtTimeStamp[z], ADR(OutDataTelegram_Module_1[2]));

			bNvAbsoluteIdx := bNvStartIndex + bObjectIndex + (aNvoSnvtTimeStampIndex[z] * bLmoCount);

			IF (FuDoNvoUpdate_Module_1(paNvoSnvtTimeStamp[z], ADR(aNvoSnvtTimeStampLast[z]), ADR(paNvoSnvtTimeStamp[z]^.bInternalUseOnly), ADR(aNvoSnvtTimeStampLast[z].bInternalUseOnly), ADR(paNvoSnvtTimeStamp[z]^.bStatusInformation), bNvAbsoluteIdx, 7, SIZEOF(aNvoSnvtTimeStampLast[z])) = FALSE) THEN
				RETURN;
			END_IF
		END_IF
	END_FOR
	FOR z := 0 TO 1 DO
		IF ((NOT FuMemCompare(ADR(aNvoSnvtAlarmLast[z]), paNvoSnvtAlarm[z], ADR(paNvoSnvtAlarm[z]^.bStatusInformation) - paNvoSnvtAlarm[z])) OR (paNvoSnvtAlarm[z]^.bStatusInformation.7 = TRUE) OR (aNvoSnvtAlarmLast[z].bInternalUseOnly.1 = TRUE)) THEN
			FuSnvtAlarmToRaw(paNvoSnvtAlarm[z], ADR(OutDataTelegram_Module_1[2]));

			bNvAbsoluteIdx := bNvStartIndex + bObjectIndex + (aNvoSnvtAlarmIndex[z] * bLmoCount);

			IF (FuDoNvoUpdate_Module_1(paNvoSnvtAlarm[z], ADR(aNvoSnvtAlarmLast[z]), ADR(paNvoSnvtAlarm[z]^.bInternalUseOnly), ADR(aNvoSnvtAlarmLast[z].bInternalUseOnly), ADR(paNvoSnvtAlarm[z]^.bStatusInformation), bNvAbsoluteIdx, 29, SIZEOF(aNvoSnvtAlarmLast[z])) = FALSE) THEN
				RETURN;
			END_IF
		END_IF
	END_FOR
	FOR z := 0 TO 3 DO
		IF ((NOT FuMemCompare(ADR(aNvoSnvtHvacModeLast[z]), paNvoSnvtHvacMode[z], ADR(paNvoSnvtHvacMode[z]^.bStatusInformation) - paNvoSnvtHvacMode[z])) OR (paNvoSnvtHvacMode[z]^.bStatusInformation.7 = TRUE) OR (aNvoSnvtHvacModeLast[z].bInternalUseOnly.1 = TRUE)) THEN
			FuSnvtHvacModeToRaw(paNvoSnvtHvacMode[z], ADR(OutDataTelegram_Module_1[2]));

			bNvAbsoluteIdx := bNvStartIndex + bObjectIndex + (aNvoSnvtHvacModeIndex[z] * bLmoCount);

			IF (FuDoNvoUpdate_Module_1(paNvoSnvtHvacMode[z], ADR(aNvoSnvtHvacModeLast[z]), ADR(paNvoSnvtHvacMode[z]^.bInternalUseOnly), ADR(aNvoSnvtHvacModeLast[z].bInternalUseOnly), ADR(paNvoSnvtHvacMode[z]^.bStatusInformation), bNvAbsoluteIdx, 1, SIZEOF(aNvoSnvtHvacModeLast[z])) = FALSE) THEN
				RETURN;
			END_IF
		END_IF
	END_FOR
	FOR z := 0 TO 3 DO
		IF ((NOT FuMemCompare(ADR(aNvoSnvtTempPLast[z]), paNvoSnvtTempP[z], ADR(paNvoSnvtTempP[z]^.bStatusInformation) - paNvoSnvtTempP[z])) OR (paNvoSnvtTempP[z]^.bStatusInformation.7 = TRUE) OR (aNvoSnvtTempPLast[z].bInternalUseOnly.1 = TRUE)) THEN
			FuSnvtTempPToRaw(paNvoSnvtTempP[z], ADR(OutDataTelegram_Module_1[2]));

			bNvAbsoluteIdx := bNvStartIndex + bObjectIndex + (aNvoSnvtTempPIndex[z] * bLmoCount);

			IF (FuDoNvoUpdate_Module_1(paNvoSnvtTempP[z], ADR(aNvoSnvtTempPLast[z]), ADR(paNvoSnvtTempP[z]^.bInternalUseOnly), ADR(aNvoSnvtTempPLast[z].bInternalUseOnly), ADR(paNvoSnvtTempP[z]^.bStatusInformation), bNvAbsoluteIdx, 2, SIZEOF(aNvoSnvtTempPLast[z])) = FALSE) THEN
				RETURN;
			END_IF
		END_IF
	END_FOR
	FOR z := 0 TO 1 DO
		IF ((NOT FuMemCompare(ADR(aNvoSnvtSwitchLast[z]), paNvoSnvtSwitch[z], ADR(paNvoSnvtSwitch[z]^.bStatusInformation) - paNvoSnvtSwitch[z])) OR (paNvoSnvtSwitch[z]^.bStatusInformation.7 = TRUE) OR (aNvoSnvtSwitchLast[z].bInternalUseOnly.1 = TRUE)) THEN
			FuSnvtSwitchToRaw(paNvoSnvtSwitch[z], ADR(OutDataTelegram_Module_1[2]));

			bNvAbsoluteIdx := bNvStartIndex + bObjectIndex + (aNvoSnvtSwitchIndex[z] * bLmoCount);

			IF (FuDoNvoUpdate_Module_1(paNvoSnvtSwitch[z], ADR(aNvoSnvtSwitchLast[z]), ADR(paNvoSnvtSwitch[z]^.bInternalUseOnly), ADR(aNvoSnvtSwitchLast[z].bInternalUseOnly), ADR(paNvoSnvtSwitch[z]^.bStatusInformation), bNvAbsoluteIdx, 2, SIZEOF(aNvoSnvtSwitchLast[z])) = FALSE) THEN
				RETURN;
			END_IF
		END_IF
	END_FOR

